//     PlcTask Inputs/GVL_iXlinker.EtherCAT_Master_EJxxxx.Beckhoff_EJ9xxx.A_0003_EJ9576_0000_0018.WcState.WcState <-> WcState/WcState
//     PlcTask Inputs/GVL_iXlinker.EtherCAT_Master_EJxxxx.Beckhoff_EJ9xxx.A_0003_EJ9576_0000_0018.WcState.InputToggle <-> WcState/InputToggle
//     PlcTask Inputs/GVL_iXlinker.EtherCAT_Master_EJxxxx.Beckhoff_EJ9xxx.A_0003_EJ9576_0000_0018.InfoData.AdsAddr <-> InfoData/AdsAddr
//     PlcTask Inputs/GVL_iXlinker.EtherCAT_Master_EJxxxx.Beckhoff_EJ9xxx.A_0003_EJ9576_0000_0018.InfoData.State <-> InfoData/State
//   PLC/PLC Instance <-> EtherCAT Master EJxxxx/Beckhoff EJ9xxx/A_0004(EJ9576-0000-0019)
//     PlcTask Inputs/GVL_iXlinker.EtherCAT_Master_EJxxxx.Beckhoff_EJ9xxx.A_0004_EJ9576_0000_0019.BCT_Inputs.Terminal_Overtemperature <-> BCT Inputs/Terminal Overtemperature
//     PlcTask Inputs/GVL_iXlinker.EtherCAT_Master_EJxxxx.Beckhoff_EJ9xxx.A_0004_EJ9576_0000_0019.BCT_Inputs.I2T_error <-> BCT Inputs/I2T error
//     PlcTask Inputs/GVL_iXlinker.EtherCAT_Master_EJxxxx.Beckhoff_EJ9xxx.A_0004_EJ9576_0000_0019.BCT_Inputs.I2T_warning <-> BCT Inputs/I2T warning
//     PlcTask Inputs/GVL_iXlinker.EtherCAT_Master_EJxxxx.Beckhoff_EJ9xxx.A_0004_EJ9576_0000_0019.BCT_Inputs.Overvoltage <-> BCT Inputs/Overvoltage
//     PlcTask Inputs/GVL_iXlinker.EtherCAT_Master_EJxxxx.Beckhoff_EJ9xxx.A_0004_EJ9576_0000_0019.BCT_Inputs.Undervoltage <-> BCT Inputs/Undervoltage
//     PlcTask Inputs/GVL_iXlinker.EtherCAT_Master_EJxxxx.Beckhoff_EJ9xxx.A_0004_EJ9576_0000_0019.BCT_Inputs.Chopper_on <-> BCT Inputs/Chopper on
//     PlcTask Inputs/GVL_iXlinker.EtherCAT_Master_EJxxxx.Beckhoff_EJ9xxx.A_0004_EJ9576_0000_0019.BCT_Inputs.Input_cycle_counter <-> BCT Inputs/Input cycle counter
//     PlcTask Inputs/GVL_iXlinker.EtherCAT_Master_EJxxxx.Beckhoff_EJ9xxx.A_0004_EJ9576_0000_0019.BCT_Inputs.DC_link_voltage <-> BCT Inputs/DC link voltage
//     PlcTask Inputs/GVL_iXlinker.EtherCAT_Master_EJxxxx.Beckhoff_EJ9xxx.A_0004_EJ9576_0000_0019.BCT_Inputs.Resistor_current <-> BCT Inputs/Resistor current
//     PlcTask Inputs/GVL_iXlinker.EtherCAT_Master_EJxxxx.Beckhoff_EJ9xxx.A_0004_EJ9576_0000_0019.BCT_Inputs.Duty_cylce <-> BCT Inputs/Duty cylce
//     PlcTask Inputs/GVL_iXlinker.EtherCAT_Master_EJxxxx.Beckhoff_EJ9xxx.A_0004_EJ9576_0000_0019.BCT_Inputs.I2T_load_factor <-> BCT Inputs/I2T load factor
//     PlcTask Inputs/GVL_iXlinker.EtherCAT_Master_EJxxxx.Beckhoff_EJ9xxx.A_0004_EJ9576_0000_0019.WcState.WcState <-> WcState/WcState
//     PlcTask Inputs/GVL_iXlinker.EtherCAT_Master_EJxxxx.Beckhoff_EJ9xxx.A_0004_EJ9576_0000_0019.WcState.InputToggle <-> WcState/InputToggle
//     PlcTask Inputs/GVL_iXlinker.EtherCAT_Master_EJxxxx.Beckhoff_EJ9xxx.A_0004_EJ9576_0000_0019.InfoData.AdsAddr <-> InfoData/AdsAddr
//     PlcTask Inputs/GVL_iXlinker.EtherCAT_Master_EJxxxx.Beckhoff_EJ9xxx.A_0004_EJ9576_0000_0019.InfoData.State <-> InfoData/State
//   PLC/PLC Instance <-> EtherCAT Master EJxxxx/Beckhoff EJ9xxx/A_0005(EJ9576-0000-0020)
//     PlcTask Inputs/GVL_iXlinker.EtherCAT_Master_EJxxxx.Beckhoff_EJ9xxx.A_0005_EJ9576_0000_0020.BCT_Inputs.Terminal_Overtemperature <-> BCT Inputs/Terminal Overtemperature
//     PlcTask Inputs/GVL_iXlinker.EtherCAT_Master_EJxxxx.Beckhoff_EJ9xxx.A_0005_EJ9576_0000_0020.BCT_Inputs.I2T_error <-> BCT Inputs/I2T error
//     PlcTask Inputs/GVL_iXlinker.EtherCAT_Master_EJxxxx.Beckhoff_EJ9xxx.A_0005_EJ9576_0000_0020.BCT_Inputs.I2T_warning <-> BCT Inputs/I2T warning
//     PlcTask Inputs/GVL_iXlinker.EtherCAT_Master_EJxxxx.Beckhoff_EJ9xxx.A_0005_EJ9576_0000_0020.BCT_Inputs.Overvoltage <-> BCT Inputs/Overvoltage
//     PlcTask Inputs/GVL_iXlinker.EtherCAT_Master_EJxxxx.Beckhoff_EJ9xxx.A_0005_EJ9576_0000_0020.BCT_Inputs.Undervoltage <-> BCT Inputs/Undervoltage
//     PlcTask Inputs/GVL_iXlinker.EtherCAT_Master_EJxxxx.Beckhoff_EJ9xxx.A_0005_EJ9576_0000_0020.BCT_Inputs.Chopper_on <-> BCT Inputs/Chopper on
//     PlcTask Inputs/GVL_iXlinker.EtherCAT_Master_EJxxxx.Beckhoff_EJ9xxx.A_0005_EJ9576_0000_0020.BCT_Inputs.Input_cycle_counter <-> BCT Inputs/Input cycle counter
//     PlcTask Inputs/GVL_iXlinker.EtherCAT_Master_EJxxxx.Beckhoff_EJ9xxx.A_0005_EJ9576_0000_0020.BCT_Inputs.DC_link_voltage <-> BCT Inputs/DC link voltage
//     PlcTask Inputs/GVL_iXlinker.EtherCAT_Master_EJxxxx.Beckhoff_EJ9xxx.A_0005_EJ9576_0000_0020.BCT_Inputs.Resistor_Current <-> BCT Inputs/Resistor Current
//     PlcTask Inputs/GVL_iXlinker.EtherCAT_Master_EJxxxx.Beckhoff_EJ9xxx.A_0005_EJ9576_0000_0020.BCT_Inputs.Duty_Cycle <-> BCT Inputs/Duty Cycle
//     PlcTask Inputs/GVL_iXlinker.EtherCAT_Master_EJxxxx.Beckhoff_EJ9xxx.A_0005_EJ9576_0000_0020.WcState.WcState <-> WcState/WcState
//     PlcTask Inputs/GVL_iXlinker.EtherCAT_Master_EJxxxx.Beckhoff_EJ9xxx.A_0005_EJ9576_0000_0020.WcState.InputToggle <-> WcState/InputToggle
//     PlcTask Inputs/GVL_iXlinker.EtherCAT_Master_EJxxxx.Beckhoff_EJ9xxx.A_0005_EJ9576_0000_0020.InfoData.AdsAddr <-> InfoData/AdsAddr
//     PlcTask Inputs/GVL_iXlinker.EtherCAT_Master_EJxxxx.Beckhoff_EJ9xxx.A_0005_EJ9576_0000_0020.InfoData.State <-> InfoData/State
//   PLC/PLC Instance <-> EtherCAT Master EJxxxx/Beckhoff EJ9xxx/A_0006(EJ9576-0000-0022)
//     PlcTask Inputs/GVL_iXlinker.EtherCAT_Master_EJxxxx.Beckhoff_EJ9xxx.A_0006_EJ9576_0000_0022.BCT_Inputs.Terminal_Overtemperature <-> BCT Inputs/Terminal Overtemperature
//     PlcTask Inputs/GVL_iXlinker.EtherCAT_Master_EJxxxx.Beckhoff_EJ9xxx.A_0006_EJ9576_0000_0022.BCT_Inputs.I2T_error <-> BCT Inputs/I2T error
//     PlcTask Inputs/GVL_iXlinker.EtherCAT_Master_EJxxxx.Beckhoff_EJ9xxx.A_0006_EJ9576_0000_0022.BCT_Inputs.I2T_warning <-> BCT Inputs/I2T warning
//     PlcTask Inputs/GVL_iXlinker.EtherCAT_Master_EJxxxx.Beckhoff_EJ9xxx.A_0006_EJ9576_0000_0022.BCT_Inputs.Overvoltage <-> BCT Inputs/Overvoltage
//     PlcTask Inputs/GVL_iXlinker.EtherCAT_Master_EJxxxx.Beckhoff_EJ9xxx.A_0006_EJ9576_0000_0022.BCT_Inputs.Undervoltage <-> BCT Inputs/Undervoltage
//     PlcTask Inputs/GVL_iXlinker.EtherCAT_Master_EJxxxx.Beckhoff_EJ9xxx.A_0006_EJ9576_0000_0022.BCT_Inputs.Chopper_on <-> BCT Inputs/Chopper on
//     PlcTask Inputs/GVL_iXlinker.EtherCAT_Master_EJxxxx.Beckhoff_EJ9xxx.A_0006_EJ9576_0000_0022.BCT_Inputs.Overcurrent_Protection <-> BCT Inputs/Overcurrent Protection
//     PlcTask Inputs/GVL_iXlinker.EtherCAT_Master_EJxxxx.Beckhoff_EJ9xxx.A_0006_EJ9576_0000_0022.BCT_Inputs.Input_cycle_counter <-> BCT Inputs/Input cycle counter
//     PlcTask Inputs/GVL_iXlinker.EtherCAT_Master_EJxxxx.Beckhoff_EJ9xxx.A_0006_EJ9576_0000_0022.BCT_Inputs.DC_link_voltage <-> BCT Inputs/DC link voltage
//     PlcTask Inputs/GVL_iXlinker.EtherCAT_Master_EJxxxx.Beckhoff_EJ9xxx.A_0006_EJ9576_0000_0022.BCT_Inputs.Resistor_Current <-> BCT Inputs/Resistor Current
//     PlcTask Inputs/GVL_iXlinker.EtherCAT_Master_EJxxxx.Beckhoff_EJ9xxx.A_0006_EJ9576_0000_0022.BCT_Inputs.Duty_Cycle <-> BCT Inputs/Duty Cycle
//     PlcTask Inputs/GVL_iXlinker.EtherCAT_Master_EJxxxx.Beckhoff_EJ9xxx.A_0006_EJ9576_0000_0022.WcState.WcState <-> WcState/WcState
//     PlcTask Inputs/GVL_iXlinker.EtherCAT_Master_EJxxxx.Beckhoff_EJ9xxx.A_0006_EJ9576_0000_0022.WcState.InputToggle <-> WcState/InputToggle
//     PlcTask Inputs/GVL_iXlinker.EtherCAT_Master_EJxxxx.Beckhoff_EJ9xxx.A_0006_EJ9576_0000_0022.InfoData.AdsAddr <-> InfoData/AdsAddr
//     PlcTask Inputs/GVL_iXlinker.EtherCAT_Master_EJxxxx.Beckhoff_EJ9xxx.A_0006_EJ9576_0000_0022.InfoData.State <-> InfoData/State
//   PLC/PLC Instance <-> EtherCAT Master EJxxxx/Beckhoff EJx9xx
//     PlcTask Inputs/GVL_iXlinker.EtherCAT_Master_EJxxxx.Beckhoff_EJx9xx.InfoData.State <-> InfoData/State
//   PLC/PLC Instance <-> EtherCAT Master EJxxxx/Beckhoff EJx9xx/Beckhoff EJx9xxEK1122
//     PlcTask Inputs/GVL_iXlinker.EtherCAT_Master_EJxxxx.Beckhoff_EJx9xx.Beckhoff_EJx9xxEK1122.InfoData.State <-> InfoData/State
//   PLC/PLC Instance <-> EtherCAT Master EJxxxx/Beckhoff EJx9xx/Beckhoff EJx9xxEK1122/Beckhoff EJx9xxsub EK1100
//     PlcTask Inputs/GVL_iXlinker.EtherCAT_Master_EJxxxx.Beckhoff_EJx9xx.Beckhoff_EJx9xxEK1122.Beckhoff_EJx9xxsub_EK1100.InfoData.State <-> InfoData/State
//   PLC/PLC Instance <-> EtherCAT Master EJxxxx/Beckhoff EJx9xx/A_0001(EJ1914-0000-0017)
//     PlcTask Inputs/GVL_iXlinker.EtherCAT_Master_EJxxxx.Beckhoff_EJx9xx.A_0001_EJ1914_0000_0017.Module_1_FSOE.FSoE_Inputs.FSOE/FSoE_Command <-> Module 1 (FSOE)/FSoE Inputs/FSOE/FSoE Command
//     PlcTask Inputs/GVL_iXlinker.EtherCAT_Master_EJxxxx.Beckhoff_EJx9xx.A_0001_EJ1914_0000_0017.Module_1_FSOE.FSoE_Inputs.FSOE/FSIN_Module_1_Channel_1_Input <-> Module 1 (FSOE)/FSoE Inputs/FSOE/FSIN Module 1.Channel 1.Input
//     PlcTask Inputs/GVL_iXlinker.EtherCAT_Master_EJxxxx.Beckhoff_EJx9xx.A_0001_EJ1914_0000_0017.Module_1_FSOE.FSoE_Inputs.FSOE/FSIN_Module_1_Channel_2_Input <-> Module 1 (FSOE)/FSoE Inputs/FSOE/FSIN Module 1.Channel 2.Input
//     PlcTask Inputs/GVL_iXlinker.EtherCAT_Master_EJxxxx.Beckhoff_EJx9xx.A_0001_EJ1914_0000_0017.Module_1_FSOE.FSoE_Inputs.FSOE/FSIN_Module_2_Channel_1_Input <-> Module 1 (FSOE)/FSoE Inputs/FSOE/FSIN Module 2.Channel 1.Input
//     PlcTask Inputs/GVL_iXlinker.EtherCAT_Master_EJxxxx.Beckhoff_EJx9xx.A_0001_EJ1914_0000_0017.Module_1_FSOE.FSoE_Inputs.FSOE/FSIN_Module_2_Channel_2_Input <-> Module 1 (FSOE)/FSoE Inputs/FSOE/FSIN Module 2.Channel 2.Input
//     PlcTask Inputs/GVL_iXlinker.EtherCAT_Master_EJxxxx.Beckhoff_EJx9xx.A_0001_EJ1914_0000_0017.Module_1_FSOE.FSoE_Inputs.FSOE/FSIN_Module_1_Module_Fault <-> Module 1 (FSOE)/FSoE Inputs/FSOE/FSIN Module 1.Module Fault
//     PlcTask Inputs/GVL_iXlinker.EtherCAT_Master_EJxxxx.Beckhoff_EJx9xx.A_0001_EJ1914_0000_0017.Module_1_FSOE.FSoE_Inputs.FSOE/FSIN_Module_2_Module_Fault <-> Module 1 (FSOE)/FSoE Inputs/FSOE/FSIN Module 2.Module Fault
//     PlcTask Inputs/GVL_iXlinker.EtherCAT_Master_EJxxxx.Beckhoff_EJx9xx.A_0001_EJ1914_0000_0017.Module_1_FSOE.FSoE_Inputs.FSOE/FSoE_CRC_000 <-> Module 1 (FSOE)/FSoE Inputs/FSOE/FSoE CRC 000
//     PlcTask Inputs/GVL_iXlinker.EtherCAT_Master_EJxxxx.Beckhoff_EJx9xx.A_0001_EJ1914_0000_0017.Module_1_FSOE.FSoE_Inputs.FSOE/FSoE_Connection_ID <-> Module 1 (FSOE)/FSoE Inputs/FSOE/FSoE Connection ID
//     PlcTask Outputs/GVL_iXlinker.EtherCAT_Master_EJxxxx.Beckhoff_EJx9xx.A_0001_EJ1914_0000_0017.Module_1_FSOE.FSoE_Outputs.FSOE/FSoE_Command <-> Module 1 (FSOE)/FSoE Outputs/FSOE/FSoE Command
//     PlcTask Outputs/GVL_iXlinker.EtherCAT_Master_EJxxxx.Beckhoff_EJx9xx.A_0001_EJ1914_0000_0017.Module_1_FSOE.FSoE_Outputs.FSOE/FSIN_Module_1_ErrAck <-> Module 1 (FSOE)/FSoE Outputs/FSOE/FSIN Module 1.ErrAck
//     PlcTask Outputs/GVL_iXlinker.EtherCAT_Master_EJxxxx.Beckhoff_EJx9xx.A_0001_EJ1914_0000_0017.Module_1_FSOE.FSoE_Outputs.FSOE/FSIN_Module_2_ErrAck <-> Module 1 (FSOE)/FSoE Outputs/FSOE/FSIN Module 2.ErrAck
//     PlcTask Outputs/GVL_iXlinker.EtherCAT_Master_EJxxxx.Beckhoff_EJx9xx.A_0001_EJ1914_0000_0017.Module_1_FSOE.FSoE_Outputs.FSOE/FSoE_CRC_000 <-> Module 1 (FSOE)/FSoE Outputs/FSOE/FSoE CRC 000
//     PlcTask Outputs/GVL_iXlinker.EtherCAT_Master_EJxxxx.Beckhoff_EJx9xx.A_0001_EJ1914_0000_0017.Module_1_FSOE.FSoE_Outputs.FSOE/FSoE_Connection_ID <-> Module 1 (FSOE)/FSoE Outputs/FSOE/FSoE Connection ID
//     PlcTask Inputs/GVL_iXlinker.EtherCAT_Master_EJxxxx.Beckhoff_EJx9xx.A_0001_EJ1914_0000_0017.Module_2_DEVICEIO.FIELDVOLTAGE_Field_Voltage_Status.Fieldvoltage_Underrange <-> Module 2 (DEVICEIO)/FIELDVOLTAGE Field Voltage Status/Fieldvoltage Underrange
//     PlcTask Inputs/GVL_iXlinker.EtherCAT_Master_EJxxxx.Beckhoff_EJx9xx.A_0001_EJ1914_0000_0017.Module_2_DEVICEIO.FIELDVOLTAGE_Field_Voltage_Status.Fieldvoltage_Overrange <-> Module 2 (DEVICEIO)/FIELDVOLTAGE Field Voltage Status/Fieldvoltage Overrange
//     PlcTask Inputs/GVL_iXlinker.EtherCAT_Master_EJxxxx.Beckhoff_EJx9xx.A_0001_EJ1914_0000_0017.Module_3_FSLOGIC.FSLOGIC_Inputs.Safe_Logic_State <-> Module 3 (FSLOGIC)/FSLOGIC Inputs/Safe Logic State
//     PlcTask Inputs/GVL_iXlinker.EtherCAT_Master_EJxxxx.Beckhoff_EJx9xx.A_0001_EJ1914_0000_0017.Module_3_FSLOGIC.FSLOGIC_Inputs.Cycle_Counter <-> Module 3 (FSLOGIC)/FSLOGIC Inputs/Cycle Counter
//     PlcTask Inputs/GVL_iXlinker.EtherCAT_Master_EJxxxx.Beckhoff_EJx9xx.A_0001_EJ1914_0000_0017.WcState.WcState <-> WcState/WcState
//     PlcTask Inputs/GVL_iXlinker.EtherCAT_Master_EJxxxx.Beckhoff_EJx9xx.A_0001_EJ1914_0000_0017.WcState.InputToggle <-> WcState/InputToggle
//     PlcTask Inputs/GVL_iXlinker.EtherCAT_Master_EJxxxx.Beckhoff_EJx9xx.A_0001_EJ1914_0000_0017.InfoData.AdsAddr <-> InfoData/AdsAddr
//     PlcTask Inputs/GVL_iXlinker.EtherCAT_Master_EJxxxx.Beckhoff_EJx9xx.A_0001_EJ1914_0000_0017.InfoData.State <-> InfoData/State
//   PLC/PLC Instance <-> EtherCAT Master EJxxxx/Beckhoff EJx9xx/A_0002(EJ1914-0000-0018)
//     PlcTask Inputs/GVL_iXlinker.EtherCAT_Master_EJxxxx.Beckhoff_EJx9xx.A_0002_EJ1914_0000_0018.Module_1_FSOE.FSoE_Inputs.FSOE/FSoE_Command <-> Module 1 (FSOE)/FSoE Inputs/FSOE/FSoE Command
//     PlcTask Inputs/GVL_iXlinker.EtherCAT_Master_EJxxxx.Beckhoff_EJx9xx.A_0002_EJ1914_0000_0018.Module_1_FSOE.FSoE_Inputs.FSOE/FSIN_Module_1_Channel_1_Input <-> Module 1 (FSOE)/FSoE Inputs/FSOE/FSIN Module 1.Channel 1.Input
//     PlcTask Inputs/GVL_iXlinker.EtherCAT_Master_EJxxxx.Beckhoff_EJx9xx.A_0002_EJ1914_0000_0018.Module_1_FSOE.FSoE_Inputs.FSOE/FSIN_Module_1_Channel_2_Input <-> Module 1 (FSOE)/FSoE Inputs/FSOE/FSIN Module 1.Channel 2.Input
//     PlcTask Inputs/GVL_iXlinker.EtherCAT_Master_EJxxxx.Beckhoff_EJx9xx.A_0002_EJ1914_0000_0018.Module_1_FSOE.FSoE_Inputs.FSOE/FSIN_Module_2_Channel_1_Input <-> Module 1 (FSOE)/FSoE Inputs/FSOE/FSIN Module 2.Channel 1.Input
//     PlcTask Inputs/GVL_iXlinker.EtherCAT_Master_EJxxxx.Beckhoff_EJx9xx.A_0002_EJ1914_0000_0018.Module_1_FSOE.FSoE_Inputs.FSOE/FSIN_Module_2_Channel_2_Input <-> Module 1 (FSOE)/FSoE Inputs/FSOE/FSIN Module 2.Channel 2.Input
//     PlcTask Inputs/GVL_iXlinker.EtherCAT_Master_EJxxxx.Beckhoff_EJx9xx.A_0002_EJ1914_0000_0018.Module_1_FSOE.FSoE_Inputs.FSOE/FSIN_Module_1_Module_Fault <-> Module 1 (FSOE)/FSoE Inputs/FSOE/FSIN Module 1.Module Fault
//     PlcTask Inputs/GVL_iXlinker.EtherCAT_Master_EJxxxx.Beckhoff_EJx9xx.A_0002_EJ1914_0000_0018.Module_1_FSOE.FSoE_Inputs.FSOE/FSIN_Module_2_Module_Fault <-> Module 1 (FSOE)/FSoE Inputs/FSOE/FSIN Module 2.Module Fault
//     PlcTask Inputs/GVL_iXlinker.EtherCAT_Master_EJxxxx.Beckhoff_EJx9xx.A_0002_EJ1914_0000_0018.Module_1_FSOE.FSoE_Inputs.FSOE/FSoE_CRC_000 <-> Module 1 (FSOE)/FSoE Inputs/FSOE/FSoE CRC 000
//     PlcTask Inputs/GVL_iXlinker.EtherCAT_Master_EJxxxx.Beckhoff_EJx9xx.A_0002_EJ1914_0000_0018.Module_1_FSOE.FSoE_Inputs.FSOE/FSoE_Connection_ID <-> Module 1 (FSOE)/FSoE Inputs/FSOE/FSoE Connection ID
//     PlcTask Outputs/GVL_iXlinker.EtherCAT_Master_EJxxxx.Beckhoff_EJx9xx.A_0002_EJ1914_0000_0018.Module_1_FSOE.FSoE_Outputs.FSOE/FSoE_Command <-> Module 1 (FSOE)/FSoE Outputs/FSOE/FSoE Command
//     PlcTask Outputs/GVL_iXlinker.EtherCAT_Master_EJxxxx.Beckhoff_EJx9xx.A_0002_EJ1914_0000_0018.Module_1_FSOE.FSoE_Outputs.FSOE/FSIN_Module_1_ErrAck <-> Module 1 (FSOE)/FSoE Outputs/FSOE/FSIN Module 1.ErrAck
//     PlcTask Outputs/GVL_iXlinker.EtherCAT_Master_EJxxxx.Beckhoff_EJx9xx.A_0002_EJ1914_0000_0018.Module_1_FSOE.FSoE_Outputs.FSOE/FSIN_Module_2_ErrAck <-> Module 1 (FSOE)/FSoE Outputs/FSOE/FSIN Module 2.ErrAck
//     PlcTask Outputs/GVL_iXlinker.EtherCAT_Master_EJxxxx.Beckhoff_EJx9xx.A_0002_EJ1914_0000_0018.Module_1_FSOE.FSoE_Outputs.FSOE/FSoE_CRC_000 <-> Module 1 (FSOE)/FSoE Outputs/FSOE/FSoE CRC 000
//     PlcTask Outputs/GVL_iXlinker.EtherCAT_Master_EJxxxx.Beckhoff_EJx9xx.A_0002_EJ1914_0000_0018.Module_1_FSOE.FSoE_Outputs.FSOE/FSoE_Connection_ID <-> Module 1 (FSOE)/FSoE Outputs/FSOE/FSoE Connection ID
//     PlcTask Inputs/GVL_iXlinker.EtherCAT_Master_EJxxxx.Beckhoff_EJx9xx.A_0002_EJ1914_0000_0018.Module_2_DEVICEIO.FIELDVOLTAGE_Field_Voltage_Status.Fieldvoltage_Underrange <-> Module 2 (DEVICEIO)/FIELDVOLTAGE Field Voltage Status/Fieldvoltage Underrange
//     PlcTask Inputs/GVL_iXlinker.EtherCAT_Master_EJxxxx.Beckhoff_EJx9xx.A_0002_EJ1914_0000_0018.Module_2_DEVICEIO.FIELDVOLTAGE_Field_Voltage_Status.Fieldvoltage_Overrange <-> Module 2 (DEVICEIO)/FIELDVOLTAGE Field Voltage Status/Fieldvoltage Overrange
//     PlcTask Inputs/GVL_iXlinker.EtherCAT_Master_EJxxxx.Beckhoff_EJx9xx.A_0002_EJ1914_0000_0018.Module_3_FSLOGIC.FSLOGIC_Inputs.Safe_Logic_State <-> Module 3 (FSLOGIC)/FSLOGIC Inputs/Safe Logic State
//     PlcTask Inputs/GVL_iXlinker.EtherCAT_Master_EJxxxx.Beckhoff_EJx9xx.A_0002_EJ1914_0000_0018.Module_3_FSLOGIC.FSLOGIC_Inputs.Cycle_Counter <-> Module 3 (FSLOGIC)/FSLOGIC Inputs/Cycle Counter
//     PlcTask Inputs/GVL_iXlinker.EtherCAT_Master_EJxxxx.Beckhoff_EJx9xx.A_0002_EJ1914_0000_0018.WcState.WcState <-> WcState/WcState
//     PlcTask Inputs/GVL_iXlinker.EtherCAT_Master_EJxxxx.Beckhoff_EJx9xx.A_0002_EJ1914_0000_0018.WcState.InputToggle <-> WcState/InputToggle
//     PlcTask Inputs/GVL_iXlinker.EtherCAT_Master_EJxxxx.Beckhoff_EJx9xx.A_0002_EJ1914_0000_0018.InfoData.AdsAddr <-> InfoData/AdsAddr
//     PlcTask Inputs/GVL_iXlinker.EtherCAT_Master_EJxxxx.Beckhoff_EJx9xx.A_0002_EJ1914_0000_0018.InfoData.State <-> InfoData/State
//   PLC/PLC Instance <-> EtherCAT Master EJxxxx/Beckhoff EJx9xx/A_0003(EJ1918-0000-0017)
//     PlcTask Inputs/GVL_iXlinker.EtherCAT_Master_EJxxxx.Beckhoff_EJx9xx.A_0003_EJ1918_0000_0017.Module_1_FSOE.FSoE_Inputs.FSOE/FSoE_Command <-> Module 1 (FSOE)/FSoE Inputs/FSOE/FSoE Command
//     PlcTask Inputs/GVL_iXlinker.EtherCAT_Master_EJxxxx.Beckhoff_EJx9xx.A_0003_EJ1918_0000_0017.Module_1_FSOE.FSoE_Inputs.FSOE/FSIN_Module_1_Channel_1_Input <-> Module 1 (FSOE)/FSoE Inputs/FSOE/FSIN Module 1.Channel 1.Input
//     PlcTask Inputs/GVL_iXlinker.EtherCAT_Master_EJxxxx.Beckhoff_EJx9xx.A_0003_EJ1918_0000_0017.Module_1_FSOE.FSoE_Inputs.FSOE/FSIN_Module_1_Channel_2_Input <-> Module 1 (FSOE)/FSoE Inputs/FSOE/FSIN Module 1.Channel 2.Input
//     PlcTask Inputs/GVL_iXlinker.EtherCAT_Master_EJxxxx.Beckhoff_EJx9xx.A_0003_EJ1918_0000_0017.Module_1_FSOE.FSoE_Inputs.FSOE/FSIN_Module_2_Channel_1_Input <-> Module 1 (FSOE)/FSoE Inputs/FSOE/FSIN Module 2.Channel 1.Input
//     PlcTask Inputs/GVL_iXlinker.EtherCAT_Master_EJxxxx.Beckhoff_EJx9xx.A_0003_EJ1918_0000_0017.Module_1_FSOE.FSoE_Inputs.FSOE/FSIN_Module_2_Channel_2_Input <-> Module 1 (FSOE)/FSoE Inputs/FSOE/FSIN Module 2.Channel 2.Input
//     PlcTask Inputs/GVL_iXlinker.EtherCAT_Master_EJxxxx.Beckhoff_EJx9xx.A_0003_EJ1918_0000_0017.Module_1_FSOE.FSoE_Inputs.FSOE/FSIN_Module_3_Channel_1_Input <-> Module 1 (FSOE)/FSoE Inputs/FSOE/FSIN Module 3.Channel 1.Input
//     PlcTask Inputs/GVL_iXlinker.EtherCAT_Master_EJxxxx.Beckhoff_EJx9xx.A_0003_EJ1918_0000_0017.Module_1_FSOE.FSoE_Inputs.FSOE/FSIN_Module_3_Channel_2_Input <-> Module 1 (FSOE)/FSoE Inputs/FSOE/FSIN Module 3.Channel 2.Input
//     PlcTask Inputs/GVL_iXlinker.EtherCAT_Master_EJxxxx.Beckhoff_EJx9xx.A_0003_EJ1918_0000_0017.Module_1_FSOE.FSoE_Inputs.FSOE/FSIN_Module_4_Channel_1_Input <-> Module 1 (FSOE)/FSoE Inputs/FSOE/FSIN Module 4.Channel 1.Input
//     PlcTask Inputs/GVL_iXlinker.EtherCAT_Master_EJxxxx.Beckhoff_EJx9xx.A_0003_EJ1918_0000_0017.Module_1_FSOE.FSoE_Inputs.FSOE/FSIN_Module_4_Channel_2_Input <-> Module 1 (FSOE)/FSoE Inputs/FSOE/FSIN Module 4.Channel 2.Input
//     PlcTask Inputs/GVL_iXlinker.EtherCAT_Master_EJxxxx.Beckhoff_EJx9xx.A_0003_EJ1918_0000_0017.Module_1_FSOE.FSoE_Inputs.FSOE/FSIN_Module_1_Module_Fault <-> Module 1 (FSOE)/FSoE Inputs/FSOE/FSIN Module 1.Module Fault
//     PlcTask Inputs/GVL_iXlinker.EtherCAT_Master_EJxxxx.Beckhoff_EJx9xx.A_0003_EJ1918_0000_0017.Module_1_FSOE.FSoE_Inputs.FSOE/FSIN_Module_2_Module_Fault <-> Module 1 (FSOE)/FSoE Inputs/FSOE/FSIN Module 2.Module Fault
//     PlcTask Inputs/GVL_iXlinker.EtherCAT_Master_EJxxxx.Beckhoff_EJx9xx.A_0003_EJ1918_0000_0017.Module_1_FSOE.FSoE_Inputs.FSOE/FSIN_Module_3_Module_Fault <-> Module 1 (FSOE)/FSoE Inputs/FSOE/FSIN Module 3.Module Fault
//     PlcTask Inputs/GVL_iXlinker.EtherCAT_Master_EJxxxx.Beckhoff_EJx9xx.A_0003_EJ1918_0000_0017.Module_1_FSOE.FSoE_Inputs.FSOE/FSIN_Module_4_Module_Fault <-> Module 1 (FSOE)/FSoE Inputs/FSOE/FSIN Module 4.Module Fault
//     PlcTask Inputs/GVL_iXlinker.EtherCAT_Master_EJxxxx.Beckhoff_EJx9xx.A_0003_EJ1918_0000_0017.Module_1_FSOE.FSoE_Inputs.FSOE/FSoE_CRC_000 <-> Module 1 (FSOE)/FSoE Inputs/FSOE/FSoE CRC 000
//     PlcTask Inputs/GVL_iXlinker.EtherCAT_Master_EJxxxx.Beckhoff_EJx9xx.A_0003_EJ1918_0000_0017.Module_1_FSOE.FSoE_Inputs.FSOE/FSoE_Connection_ID <-> Module 1 (FSOE)/FSoE Inputs/FSOE/FSoE Connection ID
//     PlcTask Outputs/GVL_iXlinker.EtherCAT_Master_EJxxxx.Beckhoff_EJx9xx.A_0003_EJ1918_0000_0017.Module_1_FSOE.FSoE_Outputs.FSOE/FSoE_Command <-> Module 1 (FSOE)/FSoE Outputs/FSOE/FSoE Command
//     PlcTask Outputs/GVL_iXlinker.EtherCAT_Master_EJxxxx.Beckhoff_EJx9xx.A_0003_EJ1918_0000_0017.Module_1_FSOE.FSoE_Outputs.FSOE/FSIN_Module_1_ErrAck <-> Module 1 (FSOE)/FSoE Outputs/FSOE/FSIN Module 1.ErrAck
//     PlcTask Outputs/GVL_iXlinker.EtherCAT_Master_EJxxxx.Beckhoff_EJx9xx.A_0003_EJ1918_0000_0017.Module_1_FSOE.FSoE_Outputs.FSOE/FSIN_Module_2_ErrAck <-> Module 1 (FSOE)/FSoE Outputs/FSOE/FSIN Module 2.ErrAck
//     PlcTask Outputs/GVL_iXlinker.EtherCAT_Master_EJxxxx.Beckhoff_EJx9xx.A_0003_EJ1918_0000_0017.Module_1_FSOE.FSoE_Outputs.FSOE/FSIN_Module_3_ErrAck <-> Module 1 (FSOE)/FSoE Outputs/FSOE/FSIN Module 3.ErrAck
//     PlcTask Outputs/GVL_iXlinker.EtherCAT_Master_EJxxxx.Beckhoff_EJx9xx.A_0003_EJ1918_0000_0017.Module_1_FSOE.FSoE_Outputs.FSOE/FSIN_Module_4_ErrAck <-> Module 1 (FSOE)/FSoE Outputs/FSOE/FSIN Module 4.ErrAck
//     PlcTask Outputs/GVL_iXlinker.EtherCAT_Master_EJxxxx.Beckhoff_EJx9xx.A_0003_EJ1918_0000_0017.Module_1_FSOE.FSoE_Outputs.FSOE/FSoE_CRC_000 <-> Module 1 (FSOE)/FSoE Outputs/FSOE/FSoE CRC 000
//     PlcTask Outputs/GVL_iXlinker.EtherCAT_Master_EJxxxx.Beckhoff_EJx9xx.A_0003_EJ1918_0000_0017.Module_1_FSOE.FSoE_Outputs.FSOE/FSoE_Connection_ID <-> Module 1 (FSOE)/FSoE Outputs/FSOE/FSoE Connection ID
//     PlcTask Inputs/GVL_iXlinker.EtherCAT_Master_EJxxxx.Beckhoff_EJx9xx.A_0003_EJ1918_0000_0017.Module_2_DEVICEIO.FIELDVOLTAGE_Field_Voltage_Status.Fieldvoltage_Underrange <-> Module 2 (DEVICEIO)/FIELDVOLTAGE Field Voltage Status/Fieldvoltage Underrange
//     PlcTask Inputs/GVL_iXlinker.EtherCAT_Master_EJxxxx.Beckhoff_EJx9xx.A_0003_EJ1918_0000_0017.Module_2_DEVICEIO.FIELDVOLTAGE_Field_Voltage_Status.Fieldvoltage_Overrange <-> Module 2 (DEVICEIO)/FIELDVOLTAGE Field Voltage Status/Fieldvoltage Overrange
//     PlcTask Inputs/GVL_iXlinker.EtherCAT_Master_EJxxxx.Beckhoff_EJx9xx.A_0003_EJ1918_0000_0017.Module_3_FSLOGIC.FSLOGIC_Inputs.Safe_Logic_State <-> Module 3 (FSLOGIC)/FSLOGIC Inputs/Safe Logic State
//     PlcTask Inputs/GVL_iXlinker.EtherCAT_Master_EJxxxx.Beckhoff_EJx9xx.A_0003_EJ1918_0000_0017.Module_3_FSLOGIC.FSLOGIC_Inputs.Cycle_Counter <-> Module 3 (FSLOGIC)/FSLOGIC Inputs/Cycle Counter
//     PlcTask Inputs/GVL_iXlinker.EtherCAT_Master_EJxxxx.Beckhoff_EJx9xx.A_0003_EJ1918_0000_0017.WcState.WcState <-> WcState/WcState
//     PlcTask Inputs/GVL_iXlinker.EtherCAT_Master_EJxxxx.Beckhoff_EJx9xx.A_0003_EJ1918_0000_0017.WcState.InputToggle <-> WcState/InputToggle
//     PlcTask Inputs/GVL_iXlinker.EtherCAT_Master_EJxxxx.Beckhoff_EJx9xx.A_0003_EJ1918_0000_0017.InfoData.AdsAddr <-> InfoData/AdsAddr
//     PlcTask Inputs/GVL_iXlinker.EtherCAT_Master_EJxxxx.Beckhoff_EJx9xx.A_0003_EJ1918_0000_0017.InfoData.State <-> InfoData/State
//   PLC/PLC Instance <-> EtherCAT Master EJxxxx/Beckhoff EJx9xx/A_0004(EJ1918-0000-0018)
//     PlcTask Inputs/GVL_iXlinker.EtherCAT_Master_EJxxxx.Beckhoff_EJx9xx.A_0004_EJ1918_0000_0018.Module_1_FSOE.FSoE_Inputs.FSOE/FSoE_Command <-> Module 1 (FSOE)/FSoE Inputs/FSOE/FSoE Command
//     PlcTask Inputs/GVL_iXlinker.EtherCAT_Master_EJxxxx.Beckhoff_EJx9xx.A_0004_EJ1918_0000_0018.Module_1_FSOE.FSoE_Inputs.FSOE/FSIN_Module_1_Channel_1_Input <-> Module 1 (FSOE)/FSoE Inputs/FSOE/FSIN Module 1.Channel 1.Input
//     PlcTask Inputs/GVL_iXlinker.EtherCAT_Master_EJxxxx.Beckhoff_EJx9xx.A_0004_EJ1918_0000_0018.Module_1_FSOE.FSoE_Inputs.FSOE/FSIN_Module_1_Channel_2_Input <-> Module 1 (FSOE)/FSoE Inputs/FSOE/FSIN Module 1.Channel 2.Input
//     PlcTask Inputs/GVL_iXlinker.EtherCAT_Master_EJxxxx.Beckhoff_EJx9xx.A_0004_EJ1918_0000_0018.Module_1_FSOE.FSoE_Inputs.FSOE/FSIN_Module_2_Channel_1_Input <-> Module 1 (FSOE)/FSoE Inputs/FSOE/FSIN Module 2.Channel 1.Input
//     PlcTask Inputs/GVL_iXlinker.EtherCAT_Master_EJxxxx.Beckhoff_EJx9xx.A_0004_EJ1918_0000_0018.Module_1_FSOE.FSoE_Inputs.FSOE/FSIN_Module_2_Channel_2_Input <-> Module 1 (FSOE)/FSoE Inputs/FSOE/FSIN Module 2.Channel 2.Input
//     PlcTask Inputs/GVL_iXlinker.EtherCAT_Master_EJxxxx.Beckhoff_EJx9xx.A_0004_EJ1918_0000_0018.Module_1_FSOE.FSoE_Inputs.FSOE/FSIN_Module_3_Channel_1_Input <-> Module 1 (FSOE)/FSoE Inputs/FSOE/FSIN Module 3.Channel 1.Input
//     PlcTask Inputs/GVL_iXlinker.EtherCAT_Master_EJxxxx.Beckhoff_EJx9xx.A_0004_EJ1918_0000_0018.Module_1_FSOE.FSoE_Inputs.FSOE/FSIN_Module_3_Channel_2_Input <-> Module 1 (FSOE)/FSoE Inputs/FSOE/FSIN Module 3.Channel 2.Input
//     PlcTask Inputs/GVL_iXlinker.EtherCAT_Master_EJxxxx.Beckhoff_EJx9xx.A_0004_EJ1918_0000_0018.Module_1_FSOE.FSoE_Inputs.FSOE/FSIN_Module_4_Channel_1_Input <-> Module 1 (FSOE)/FSoE Inputs/FSOE/FSIN Module 4.Channel 1.Input
//     PlcTask Inputs/GVL_iXlinker.EtherCAT_Master_EJxxxx.Beckhoff_EJx9xx.A_0004_EJ1918_0000_0018.Module_1_FSOE.FSoE_Inputs.FSOE/FSIN_Module_4_Channel_2_Input <-> Module 1 (FSOE)/FSoE Inputs/FSOE/FSIN Module 4.Channel 2.Input
//     PlcTask Inputs/GVL_iXlinker.EtherCAT_Master_EJxxxx.Beckhoff_EJx9xx.A_0004_EJ1918_0000_0018.Module_1_FSOE.FSoE_Inputs.FSOE/FSIN_Module_1_Module_Fault <-> Module 1 (FSOE)/FSoE Inputs/FSOE/FSIN Module 1.Module Fault
//     PlcTask Inputs/GVL_iXlinker.EtherCAT_Master_EJxxxx.Beckhoff_EJx9xx.A_0004_EJ1918_0000_0018.Module_1_FSOE.FSoE_Inputs.FSOE/FSIN_Module_2_Module_Fault <-> Module 1 (FSOE)/FSoE Inputs/FSOE/FSIN Module 2.Module Fault
//     PlcTask Inputs/GVL_iXlinker.EtherCAT_Master_EJxxxx.Beckhoff_EJx9xx.A_0004_EJ1918_0000_0018.Module_1_FSOE.FSoE_Inputs.FSOE/FSIN_Module_3_Module_Fault <-> Module 1 (FSOE)/FSoE Inputs/FSOE/FSIN Module 3.Module Fault
//     PlcTask Inputs/GVL_iXlinker.EtherCAT_Master_EJxxxx.Beckhoff_EJx9xx.A_0004_EJ1918_0000_0018.Module_1_FSOE.FSoE_Inputs.FSOE/FSIN_Module_4_Module_Fault <-> Module 1 (FSOE)/FSoE Inputs/FSOE/FSIN Module 4.Module Fault
//     PlcTask Inputs/GVL_iXlinker.EtherCAT_Master_EJxxxx.Beckhoff_EJx9xx.A_0004_EJ1918_0000_0018.Module_1_FSOE.FSoE_Inputs.FSOE/FSoE_CRC_000 <-> Module 1 (FSOE)/FSoE Inputs/FSOE/FSoE CRC 000
//     PlcTask Inputs/GVL_iXlinker.EtherCAT_Master_EJxxxx.Beckhoff_EJx9xx.A_0004_EJ1918_0000_0018.Module_1_FSOE.FSoE_Inputs.FSOE/FSoE_Connection_ID <-> Module 1 (FSOE)/FSoE Inputs/FSOE/FSoE Connection ID
//     PlcTask Outputs/GVL_iXlinker.EtherCAT_Master_EJxxxx.Beckhoff_EJx9xx.A_0004_EJ1918_0000_0018.Module_1_FSOE.FSoE_Outputs.FSOE/FSoE_Command <-> Module 1 (FSOE)/FSoE Outputs/FSOE/FSoE Command
//     PlcTask Outputs/GVL_iXlinker.EtherCAT_Master_EJxxxx.Beckhoff_EJx9xx.A_0004_EJ1918_0000_0018.Module_1_FSOE.FSoE_Outputs.FSOE/FSIN_Module_1_ErrAck <-> Module 1 (FSOE)/FSoE Outputs/FSOE/FSIN Module 1.ErrAck
//     PlcTask Outputs/GVL_iXlinker.EtherCAT_Master_EJxxxx.Beckhoff_EJx9xx.A_0004_EJ1918_0000_0018.Module_1_FSOE.FSoE_Outputs.FSOE/FSIN_Module_2_ErrAck <-> Module 1 (FSOE)/FSoE Outputs/FSOE/FSIN Module 2.ErrAck
//     PlcTask Outputs/GVL_iXlinker.EtherCAT_Master_EJxxxx.Beckhoff_EJx9xx.A_0004_EJ1918_0000_0018.Module_1_FSOE.FSoE_Outputs.FSOE/FSIN_Module_3_ErrAck <-> Module 1 (FSOE)/FSoE Outputs/FSOE/FSIN Module 3.ErrAck
//     PlcTask Outputs/GVL_iXlinker.EtherCAT_Master_EJxxxx.Beckhoff_EJx9xx.A_0004_EJ1918_0000_0018.Module_1_FSOE.FSoE_Outputs.FSOE/FSIN_Module_4_ErrAck <-> Module 1 (FSOE)/FSoE Outputs/FSOE/FSIN Module 4.ErrAck
//     PlcTask Outputs/GVL_iXlinker.EtherCAT_Master_EJxxxx.Beckhoff_EJx9xx.A_0004_EJ1918_0000_0018.Module_1_FSOE.FSoE_Outputs.FSOE/FSoE_CRC_000 <-> Module 1 (FSOE)/FSoE Outputs/FSOE/FSoE CRC 000
//     PlcTask Outputs/GVL_iXlinker.EtherCAT_Master_EJxxxx.Beckhoff_EJx9xx.A_0004_EJ1918_0000_0018.Module_1_FSOE.FSoE_Outputs.FSOE/FSoE_Connection_ID <-> Module 1 (FSOE)/FSoE Outputs/FSOE/FSoE Connection ID
//     PlcTask Inputs/GVL_iXlinker.EtherCAT_Master_EJxxxx.Beckhoff_EJx9xx.A_0004_EJ1918_0000_0018.Module_2_DEVICEIO.FIELDVOLTAGE_Field_Voltage_Status.Fieldvoltage_Underrange <-> Module 2 (DEVICEIO)/FIELDVOLTAGE Field Voltage Status/Fieldvoltage Underrange
//     PlcTask Inputs/GVL_iXlinker.EtherCAT_Master_EJxxxx.Beckhoff_EJx9xx.A_0004_EJ1918_0000_0018.Module_2_DEVICEIO.FIELDVOLTAGE_Field_Voltage_Status.Fieldvoltage_Overrange <-> Module 2 (DEVICEIO)/FIELDVOLTAGE Field Voltage Status/Fieldvoltage Overrange
//     PlcTask Inputs/GVL_iXlinker.EtherCAT_Master_EJxxxx.Beckhoff_EJx9xx.A_0004_EJ1918_0000_0018.Module_3_FSLOGIC.FSLOGIC_Inputs.Safe_Logic_State <-> Module 3 (FSLOGIC)/FSLOGIC Inputs/Safe Logic State
//     PlcTask Inputs/GVL_iXlinker.EtherCAT_Master_EJxxxx.Beckhoff_EJx9xx.A_0004_EJ1918_0000_0018.Module_3_FSLOGIC.FSLOGIC_Inputs.Cycle_Counter <-> Module 3 (FSLOGIC)/FSLOGIC Inputs/Cycle Counter
//     PlcTask Inputs/GVL_iXlinker.EtherCAT_Master_EJxxxx.Beckhoff_EJx9xx.A_0004_EJ1918_0000_0018.WcState.WcState <-> WcState/WcState
//     PlcTask Inputs/GVL_iXlinker.EtherCAT_Master_EJxxxx.Beckhoff_EJx9xx.A_0004_EJ1918_0000_0018.WcState.InputToggle <-> WcState/InputToggle
//     PlcTask Inputs/GVL_iXlinker.EtherCAT_Master_EJxxxx.Beckhoff_EJx9xx.A_0004_EJ1918_0000_0018.InfoData.AdsAddr <-> InfoData/AdsAddr
//     PlcTask Inputs/GVL_iXlinker.EtherCAT_Master_EJxxxx.Beckhoff_EJx9xx.A_0004_EJ1918_0000_0018.InfoData.State <-> InfoData/State
//   PLC/PLC Instance <-> EtherCAT Master EJxxxx/Beckhoff EJx9xx/A_0005(EJ1957-0000-0017)
//     PlcTask Inputs/GVL_iXlinker.EtherCAT_Master_EJxxxx.Beckhoff_EJx9xx.A_0005_EJ1957_0000_0017.Module_1_FSOE.FSoE_Inputs.FSOE/FSoE_Command <-> Module 1 (FSOE)/FSoE Inputs/FSOE/FSoE Command
//     PlcTask Inputs/GVL_iXlinker.EtherCAT_Master_EJxxxx.Beckhoff_EJx9xx.A_0005_EJ1957_0000_0017.Module_1_FSOE.FSoE_Inputs.FSOE/FSOUT_Module_Module_Fault <-> Module 1 (FSOE)/FSoE Inputs/FSOE/FSOUT Module.Module Fault
//     PlcTask Inputs/GVL_iXlinker.EtherCAT_Master_EJxxxx.Beckhoff_EJx9xx.A_0005_EJ1957_0000_0017.Module_1_FSOE.FSoE_Inputs.FSOE/FSIN_Module_1_Channel_1_Input <-> Module 1 (FSOE)/FSoE Inputs/FSOE/FSIN Module 1.Channel 1.Input
//     PlcTask Inputs/GVL_iXlinker.EtherCAT_Master_EJxxxx.Beckhoff_EJx9xx.A_0005_EJ1957_0000_0017.Module_1_FSOE.FSoE_Inputs.FSOE/FSIN_Module_1_Channel_2_Input <-> Module 1 (FSOE)/FSoE Inputs/FSOE/FSIN Module 1.Channel 2.Input
//     PlcTask Inputs/GVL_iXlinker.EtherCAT_Master_EJxxxx.Beckhoff_EJx9xx.A_0005_EJ1957_0000_0017.Module_1_FSOE.FSoE_Inputs.FSOE/FSIN_Module_2_Channel_1_Input <-> Module 1 (FSOE)/FSoE Inputs/FSOE/FSIN Module 2.Channel 1.Input
//     PlcTask Inputs/GVL_iXlinker.EtherCAT_Master_EJxxxx.Beckhoff_EJx9xx.A_0005_EJ1957_0000_0017.Module_1_FSOE.FSoE_Inputs.FSOE/FSIN_Module_2_Channel_2_Input <-> Module 1 (FSOE)/FSoE Inputs/FSOE/FSIN Module 2.Channel 2.Input
//     PlcTask Inputs/GVL_iXlinker.EtherCAT_Master_EJxxxx.Beckhoff_EJx9xx.A_0005_EJ1957_0000_0017.Module_1_FSOE.FSoE_Inputs.FSOE/FSIN_Module_3_Channel_1_Input <-> Module 1 (FSOE)/FSoE Inputs/FSOE/FSIN Module 3.Channel 1.Input
//     PlcTask Inputs/GVL_iXlinker.EtherCAT_Master_EJxxxx.Beckhoff_EJx9xx.A_0005_EJ1957_0000_0017.Module_1_FSOE.FSoE_Inputs.FSOE/FSIN_Module_3_Channel_2_Input <-> Module 1 (FSOE)/FSoE Inputs/FSOE/FSIN Module 3.Channel 2.Input
//     PlcTask Inputs/GVL_iXlinker.EtherCAT_Master_EJxxxx.Beckhoff_EJx9xx.A_0005_EJ1957_0000_0017.Module_1_FSOE.FSoE_Inputs.FSOE/FSIN_Module_4_Channel_1_Input <-> Module 1 (FSOE)/FSoE Inputs/FSOE/FSIN Module 4.Channel 1.Input
//     PlcTask Inputs/GVL_iXlinker.EtherCAT_Master_EJxxxx.Beckhoff_EJx9xx.A_0005_EJ1957_0000_0017.Module_1_FSOE.FSoE_Inputs.FSOE/FSIN_Module_4_Channel_2_Input <-> Module 1 (FSOE)/FSoE Inputs/FSOE/FSIN Module 4.Channel 2.Input
//     PlcTask Inputs/GVL_iXlinker.EtherCAT_Master_EJxxxx.Beckhoff_EJx9xx.A_0005_EJ1957_0000_0017.Module_1_FSOE.FSoE_Inputs.FSOE/FSIN_Module_1_Module_Fault <-> Module 1 (FSOE)/FSoE Inputs/FSOE/FSIN Module 1.Module Fault
//     PlcTask Inputs/GVL_iXlinker.EtherCAT_Master_EJxxxx.Beckhoff_EJx9xx.A_0005_EJ1957_0000_0017.Module_1_FSOE.FSoE_Inputs.FSOE/FSIN_Module_2_Module_Fault <-> Module 1 (FSOE)/FSoE Inputs/FSOE/FSIN Module 2.Module Fault
//     PlcTask Inputs/GVL_iXlinker.EtherCAT_Master_EJxxxx.Beckhoff_EJx9xx.A_0005_EJ1957_0000_0017.Module_1_FSOE.FSoE_Inputs.FSOE/FSIN_Module_3_Module_Fault <-> Module 1 (FSOE)/FSoE Inputs/FSOE/FSIN Module 3.Module Fault
//     PlcTask Inputs/GVL_iXlinker.EtherCAT_Master_EJxxxx.Beckhoff_EJx9xx.A_0005_EJ1957_0000_0017.Module_1_FSOE.FSoE_Inputs.FSOE/FSIN_Module_4_Module_Fault <-> Module 1 (FSOE)/FSoE Inputs/FSOE/FSIN Module 4.Module Fault
//     PlcTask Inputs/GVL_iXlinker.EtherCAT_Master_EJxxxx.Beckhoff_EJx9xx.A_0005_EJ1957_0000_0017.Module_1_FSOE.FSoE_Inputs.FSOE/FSoE_CRC_000 <-> Module 1 (FSOE)/FSoE Inputs/FSOE/FSoE CRC 000
//     PlcTask Inputs/GVL_iXlinker.EtherCAT_Master_EJxxxx.Beckhoff_EJx9xx.A_0005_EJ1957_0000_0017.Module_1_FSOE.FSoE_Inputs.FSOE/FSoE_Connection_ID <-> Module 1 (FSOE)/FSoE Inputs/FSOE/FSoE Connection ID
//     PlcTask Outputs/GVL_iXlinker.EtherCAT_Master_EJxxxx.Beckhoff_EJx9xx.A_0005_EJ1957_0000_0017.Module_1_FSOE.FSoE_Outputs.FSOE/FSoE_Command <-> Module 1 (FSOE)/FSoE Outputs/FSOE/FSoE Command
//     PlcTask Outputs/GVL_iXlinker.EtherCAT_Master_EJxxxx.Beckhoff_EJx9xx.A_0005_EJ1957_0000_0017.Module_1_FSOE.FSoE_Outputs.FSOE/FSOUT_Module_Channel_1_Output <-> Module 1 (FSOE)/FSoE Outputs/FSOE/FSOUT Module.Channel 1.Output
//     PlcTask Outputs/GVL_iXlinker.EtherCAT_Master_EJxxxx.Beckhoff_EJx9xx.A_0005_EJ1957_0000_0017.Module_1_FSOE.FSoE_Outputs.FSOE/FSOUT_Module_Channel_2_Output <-> Module 1 (FSOE)/FSoE Outputs/FSOE/FSOUT Module.Channel 2.Output
//     PlcTask Outputs/GVL_iXlinker.EtherCAT_Master_EJxxxx.Beckhoff_EJx9xx.A_0005_EJ1957_0000_0017.Module_1_FSOE.FSoE_Outputs.FSOE/FSOUT_Module_Channel_3_Output <-> Module 1 (FSOE)/FSoE Outputs/FSOE/FSOUT Module.Channel 3.Output
//     PlcTask Outputs/GVL_iXlinker.EtherCAT_Master_EJxxxx.Beckhoff_EJx9xx.A_0005_EJ1957_0000_0017.Module_1_FSOE.FSoE_Outputs.FSOE/FSOUT_Module_Channel_4_Output <-> Module 1 (FSOE)/FSoE Outputs/FSOE/FSOUT Module.Channel 4.Output
//     PlcTask Outputs/GVL_iXlinker.EtherCAT_Master_EJxxxx.Beckhoff_EJx9xx.A_0005_EJ1957_0000_0017.Module_1_FSOE.FSoE_Outputs.FSOE/FSOUT_Module_ErrAck <-> Module 1 (FSOE)/FSoE Outputs/FSOE/FSOUT Module.ErrAck
//     PlcTask Outputs/GVL_iXlinker.EtherCAT_Master_EJxxxx.Beckhoff_EJx9xx.A_0005_EJ1957_0000_0017.Module_1_FSOE.FSoE_Outputs.FSOE/FSIN_Module_1_ErrAck <-> Module 1 (FSOE)/FSoE Outputs/FSOE/FSIN Module 1.ErrAck
//     PlcTask Outputs/GVL_iXlinker.EtherCAT_Master_EJxxxx.Beckhoff_EJx9xx.A_0005_EJ1957_0000_0017.Module_1_FSOE.FSoE_Outputs.FSOE/FSIN_Module_2_ErrAck <-> Module 1 (FSOE)/FSoE Outputs/FSOE/FSIN Module 2.ErrAck
//     PlcTask Outputs/GVL_iXlinker.EtherCAT_Master_EJxxxx.Beckhoff_EJx9xx.A_0005_EJ1957_0000_0017.Module_1_FSOE.FSoE_Outputs.FSOE/FSIN_Module_3_ErrAck <-> Module 1 (FSOE)/FSoE Outputs/FSOE/FSIN Module 3.ErrAck
//     PlcTask Outputs/GVL_iXlinker.EtherCAT_Master_EJxxxx.Beckhoff_EJx9xx.A_0005_EJ1957_0000_0017.Module_1_FSOE.FSoE_Outputs.FSOE/FSIN_Module_4_ErrAck <-> Module 1 (FSOE)/FSoE Outputs/FSOE/FSIN Module 4.ErrAck
//     PlcTask Outputs/GVL_iXlinker.EtherCAT_Master_EJxxxx.Beckhoff_EJx9xx.A_0005_EJ1957_0000_0017.Module_1_FSOE.FSoE_Outputs.FSOE/FSoE_CRC_000 <-> Module 1 (FSOE)/FSoE Outputs/FSOE/FSoE CRC 000
//     PlcTask Outputs/GVL_iXlinker.EtherCAT_Master_EJxxxx.Beckhoff_EJx9xx.A_0005_EJ1957_0000_0017.Module_1_FSOE.FSoE_Outputs.FSOE/FSoE_Connection_ID <-> Module 1 (FSOE)/FSoE Outputs/FSOE/FSoE Connection ID
//     PlcTask Outputs/GVL_iXlinker.EtherCAT_Master_EJxxxx.Beckhoff_EJx9xx.A_0005_EJ1957_0000_0017.Module_2_FSOUT.Outputs.Channel_1_Standard_Output <-> Module 2 (FSOUT)/Outputs/Channel 1.Standard Output
//     PlcTask Outputs/GVL_iXlinker.EtherCAT_Master_EJxxxx.Beckhoff_EJx9xx.A_0005_EJ1957_0000_0017.Module_2_FSOUT.Outputs.Channel_2_Standard_Output <-> Module 2 (FSOUT)/Outputs/Channel 2.Standard Output
//     PlcTask Outputs/GVL_iXlinker.EtherCAT_Master_EJxxxx.Beckhoff_EJx9xx.A_0005_EJ1957_0000_0017.Module_2_FSOUT.Outputs.Channel_3_Standard_Output <-> Module 2 (FSOUT)/Outputs/Channel 3.Standard Output
//     PlcTask Outputs/GVL_iXlinker.EtherCAT_Master_EJxxxx.Beckhoff_EJx9xx.A_0005_EJ1957_0000_0017.Module_2_FSOUT.Outputs.Channel_4_Standard_Output <-> Module 2 (FSOUT)/Outputs/Channel 4.Standard Output
//     PlcTask Inputs/GVL_iXlinker.EtherCAT_Master_EJxxxx.Beckhoff_EJx9xx.A_0005_EJ1957_0000_0017.Module_3_DEVICEIO.FIELDVOLTAGE_Field_Voltage_Status.Fieldvoltage_Underrange <-> Module 3 (DEVICEIO)/FIELDVOLTAGE Field Voltage Status/Fieldvoltage Underrange
//     PlcTask Inputs/GVL_iXlinker.EtherCAT_Master_EJxxxx.Beckhoff_EJx9xx.A_0005_EJ1957_0000_0017.Module_3_DEVICEIO.FIELDVOLTAGE_Field_Voltage_Status.Fieldvoltage_Overrange <-> Module 3 (DEVICEIO)/FIELDVOLTAGE Field Voltage Status/Fieldvoltage Overrange
//     PlcTask Inputs/GVL_iXlinker.EtherCAT_Master_EJxxxx.Beckhoff_EJx9xx.A_0005_EJ1957_0000_0017.Module_4_FSLOGIC.FSLOGIC_Inputs.Safe_Logic_State <-> Module 4 (FSLOGIC)/FSLOGIC Inputs/Safe Logic State
//     PlcTask Inputs/GVL_iXlinker.EtherCAT_Master_EJxxxx.Beckhoff_EJx9xx.A_0005_EJ1957_0000_0017.Module_4_FSLOGIC.FSLOGIC_Inputs.Cycle_Counter <-> Module 4 (FSLOGIC)/FSLOGIC Inputs/Cycle Counter
//     PlcTask Inputs/GVL_iXlinker.EtherCAT_Master_EJxxxx.Beckhoff_EJx9xx.A_0005_EJ1957_0000_0017.WcState.WcState0 <-> WcState/WcState0
//     PlcTask Inputs/GVL_iXlinker.EtherCAT_Master_EJxxxx.Beckhoff_EJx9xx.A_0005_EJ1957_0000_0017.WcState.WcState1 <-> WcState/WcState1
//     PlcTask Inputs/GVL_iXlinker.EtherCAT_Master_EJxxxx.Beckhoff_EJx9xx.A_0005_EJ1957_0000_0017.WcState.InputToggle0 <-> WcState/InputToggle0
//     PlcTask Inputs/GVL_iXlinker.EtherCAT_Master_EJxxxx.Beckhoff_EJx9xx.A_0005_EJ1957_0000_0017.WcState.InputToggle1 <-> WcState/InputToggle1
//     PlcTask Inputs/GVL_iXlinker.EtherCAT_Master_EJxxxx.Beckhoff_EJx9xx.A_0005_EJ1957_0000_0017.InfoData.AdsAddr <-> InfoData/AdsAddr
//     PlcTask Inputs/GVL_iXlinker.EtherCAT_Master_EJxxxx.Beckhoff_EJx9xx.A_0005_EJ1957_0000_0017.InfoData.State <-> InfoData/State
//   PLC/PLC Instance <-> EtherCAT Master EJxxxx/Beckhoff EJx9xx/A_0006(EJ1957-0000-0018)
//     PlcTask Inputs/GVL_iXlinker.EtherCAT_Master_EJxxxx.Beckhoff_EJx9xx.A_0006_EJ1957_0000_0018.Module_1_FSOE.FSoE_Inputs.FSOE/FSoE_Command <-> Module 1 (FSOE)/FSoE Inputs/FSOE/FSoE Command
//     PlcTask Inputs/GVL_iXlinker.EtherCAT_Master_EJxxxx.Beckhoff_EJx9xx.A_0006_EJ1957_0000_0018.Module_1_FSOE.FSoE_Inputs.FSOE/FSOUT_Module_Module_Fault <-> Module 1 (FSOE)/FSoE Inputs/FSOE/FSOUT Module.Module Fault
//     PlcTask Inputs/GVL_iXlinker.EtherCAT_Master_EJxxxx.Beckhoff_EJx9xx.A_0006_EJ1957_0000_0018.Module_1_FSOE.FSoE_Inputs.FSOE/FSIN_Module_1_Channel_1_Input <-> Module 1 (FSOE)/FSoE Inputs/FSOE/FSIN Module 1.Channel 1.Input
//     PlcTask Inputs/GVL_iXlinker.EtherCAT_Master_EJxxxx.Beckhoff_EJx9xx.A_0006_EJ1957_0000_0018.Module_1_FSOE.FSoE_Inputs.FSOE/FSIN_Module_1_Channel_2_Input <-> Module 1 (FSOE)/FSoE Inputs/FSOE/FSIN Module 1.Channel 2.Input
//     PlcTask Inputs/GVL_iXlinker.EtherCAT_Master_EJxxxx.Beckhoff_EJx9xx.A_0006_EJ1957_0000_0018.Module_1_FSOE.FSoE_Inputs.FSOE/FSIN_Module_2_Channel_1_Input <-> Module 1 (FSOE)/FSoE Inputs/FSOE/FSIN Module 2.Channel 1.Input
//     PlcTask Inputs/GVL_iXlinker.EtherCAT_Master_EJxxxx.Beckhoff_EJx9xx.A_0006_EJ1957_0000_0018.Module_1_FSOE.FSoE_Inputs.FSOE/FSIN_Module_2_Channel_2_Input <-> Module 1 (FSOE)/FSoE Inputs/FSOE/FSIN Module 2.Channel 2.Input
//     PlcTask Inputs/GVL_iXlinker.EtherCAT_Master_EJxxxx.Beckhoff_EJx9xx.A_0006_EJ1957_0000_0018.Module_1_FSOE.FSoE_Inputs.FSOE/FSIN_Module_3_Channel_1_Input <-> Module 1 (FSOE)/FSoE Inputs/FSOE/FSIN Module 3.Channel 1.Input
//     PlcTask Inputs/GVL_iXlinker.EtherCAT_Master_EJxxxx.Beckhoff_EJx9xx.A_0006_EJ1957_0000_0018.Module_1_FSOE.FSoE_Inputs.FSOE/FSIN_Module_3_Channel_2_Input <-> Module 1 (FSOE)/FSoE Inputs/FSOE/FSIN Module 3.Channel 2.Input
//     PlcTask Inputs/GVL_iXlinker.EtherCAT_Master_EJxxxx.Beckhoff_EJx9xx.A_0006_EJ1957_0000_0018.Module_1_FSOE.FSoE_Inputs.FSOE/FSIN_Module_4_Channel_1_Input <-> Module 1 (FSOE)/FSoE Inputs/FSOE/FSIN Module 4.Channel 1.Input
//     PlcTask Inputs/GVL_iXlinker.EtherCAT_Master_EJxxxx.Beckhoff_EJx9xx.A_0006_EJ1957_0000_0018.Module_1_FSOE.FSoE_Inputs.FSOE/FSIN_Module_4_Channel_2_Input <-> Module 1 (FSOE)/FSoE Inputs/FSOE/FSIN Module 4.Channel 2.Input
//     PlcTask Inputs/GVL_iXlinker.EtherCAT_Master_EJxxxx.Beckhoff_EJx9xx.A_0006_EJ1957_0000_0018.Module_1_FSOE.FSoE_Inputs.FSOE/FSIN_Module_1_Module_Fault <-> Module 1 (FSOE)/FSoE Inputs/FSOE/FSIN Module 1.Module Fault
//     PlcTask Inputs/GVL_iXlinker.EtherCAT_Master_EJxxxx.Beckhoff_EJx9xx.A_0006_EJ1957_0000_0018.Module_1_FSOE.FSoE_Inputs.FSOE/FSIN_Module_2_Module_Fault <-> Module 1 (FSOE)/FSoE Inputs/FSOE/FSIN Module 2.Module Fault
//     PlcTask Inputs/GVL_iXlinker.EtherCAT_Master_EJxxxx.Beckhoff_EJx9xx.A_0006_EJ1957_0000_0018.Module_1_FSOE.FSoE_Inputs.FSOE/FSIN_Module_3_Module_Fault <-> Module 1 (FSOE)/FSoE Inputs/FSOE/FSIN Module 3.Module Fault
//     PlcTask Inputs/GVL_iXlinker.EtherCAT_Master_EJxxxx.Beckhoff_EJx9xx.A_0006_EJ1957_0000_0018.Module_1_FSOE.FSoE_Inputs.FSOE/FSIN_Module_4_Module_Fault <-> Module 1 (FSOE)/FSoE Inputs/FSOE/FSIN Module 4.Module Fault
//     PlcTask Inputs/GVL_iXlinker.EtherCAT_Master_EJxxxx.Beckhoff_EJx9xx.A_0006_EJ1957_0000_0018.Module_1_FSOE.FSoE_Inputs.FSOE/FSoE_CRC_000 <-> Module 1 (FSOE)/FSoE Inputs/FSOE/FSoE CRC 000
//     PlcTask Inputs/GVL_iXlinker.EtherCAT_Master_EJxxxx.Beckhoff_EJx9xx.A_0006_EJ1957_0000_0018.Module_1_FSOE.FSoE_Inputs.FSOE/FSoE_Connection_ID <-> Module 1 (FSOE)/FSoE Inputs/FSOE/FSoE Connection ID
//     PlcTask Outputs/GVL_iXlinker.EtherCAT_Master_EJxxxx.Beckhoff_EJx9xx.A_0006_EJ1957_0000_0018.Module_1_FSOE.FSoE_Outputs.FSOE/FSoE_Command <-> Module 1 (FSOE)/FSoE Outputs/FSOE/FSoE Command
//     PlcTask Outputs/GVL_iXlinker.EtherCAT_Master_EJxxxx.Beckhoff_EJx9xx.A_0006_EJ1957_0000_0018.Module_1_FSOE.FSoE_Outputs.FSOE/FSOUT_Module_Channel_1_Output <-> Module 1 (FSOE)/FSoE Outputs/FSOE/FSOUT Module.Channel 1.Output
//     PlcTask Outputs/GVL_iXlinker.EtherCAT_Master_EJxxxx.Beckhoff_EJx9xx.A_0006_EJ1957_0000_0018.Module_1_FSOE.FSoE_Outputs.FSOE/FSOUT_Module_Channel_2_Output <-> Module 1 (FSOE)/FSoE Outputs/FSOE/FSOUT Module.Channel 2.Output
//     PlcTask Outputs/GVL_iXlinker.EtherCAT_Master_EJxxxx.Beckhoff_EJx9xx.A_0006_EJ1957_0000_0018.Module_1_FSOE.FSoE_Outputs.FSOE/FSOUT_Module_Channel_3_Output <-> Module 1 (FSOE)/FSoE Outputs/FSOE/FSOUT Module.Channel 3.Output
//     PlcTask Outputs/GVL_iXlinker.EtherCAT_Master_EJxxxx.Beckhoff_EJx9xx.A_0006_EJ1957_0000_0018.Module_1_FSOE.FSoE_Outputs.FSOE/FSOUT_Module_Channel_4_Output <-> Module 1 (FSOE)/FSoE Outputs/FSOE/FSOUT Module.Channel 4.Output
//     PlcTask Outputs/GVL_iXlinker.EtherCAT_Master_EJxxxx.Beckhoff_EJx9xx.A_0006_EJ1957_0000_0018.Module_1_FSOE.FSoE_Outputs.FSOE/FSOUT_Module_ErrAck <-> Module 1 (FSOE)/FSoE Outputs/FSOE/FSOUT Module.ErrAck
//     PlcTask Outputs/GVL_iXlinker.EtherCAT_Master_EJxxxx.Beckhoff_EJx9xx.A_0006_EJ1957_0000_0018.Module_1_FSOE.FSoE_Outputs.FSOE/FSIN_Module_1_ErrAck <-> Module 1 (FSOE)/FSoE Outputs/FSOE/FSIN Module 1.ErrAck
//     PlcTask Outputs/GVL_iXlinker.EtherCAT_Master_EJxxxx.Beckhoff_EJx9xx.A_0006_EJ1957_0000_0018.Module_1_FSOE.FSoE_Outputs.FSOE/FSIN_Module_2_ErrAck <-> Module 1 (FSOE)/FSoE Outputs/FSOE/FSIN Module 2.ErrAck
//     PlcTask Outputs/GVL_iXlinker.EtherCAT_Master_EJxxxx.Beckhoff_EJx9xx.A_0006_EJ1957_0000_0018.Module_1_FSOE.FSoE_Outputs.FSOE/FSIN_Module_3_ErrAck <-> Module 1 (FSOE)/FSoE Outputs/FSOE/FSIN Module 3.ErrAck
//     PlcTask Outputs/GVL_iXlinker.EtherCAT_Master_EJxxxx.Beckhoff_EJx9xx.A_0006_EJ1957_0000_0018.Module_1_FSOE.FSoE_Outputs.FSOE/FSIN_Module_4_ErrAck <-> Module 1 (FSOE)/FSoE Outputs/FSOE/FSIN Module 4.ErrAck
//     PlcTask Outputs/GVL_iXlinker.EtherCAT_Master_EJxxxx.Beckhoff_EJx9xx.A_0006_EJ1957_0000_0018.Module_1_FSOE.FSoE_Outputs.FSOE/FSoE_CRC_000 <-> Module 1 (FSOE)/FSoE Outputs/FSOE/FSoE CRC 000
//     PlcTask Outputs/GVL_iXlinker.EtherCAT_Master_EJxxxx.Beckhoff_EJx9xx.A_0006_EJ1957_0000_0018.Module_1_FSOE.FSoE_Outputs.FSOE/FSoE_Connection_ID <-> Module 1 (FSOE)/FSoE Outputs/FSOE/FSoE Connection ID
//     PlcTask Outputs/GVL_iXlinker.EtherCAT_Master_EJxxxx.Beckhoff_EJx9xx.A_0006_EJ1957_0000_0018.Module_2_FSOUT.Outputs.Channel_1_Standard_Output <-> Module 2 (FSOUT)/Outputs/Channel 1.Standard Output
//     PlcTask Outputs/GVL_iXlinker.EtherCAT_Master_EJxxxx.Beckhoff_EJx9xx.A_0006_EJ1957_0000_0018.Module_2_FSOUT.Outputs.Channel_2_Standard_Output <-> Module 2 (FSOUT)/Outputs/Channel 2.Standard Output
//     PlcTask Outputs/GVL_iXlinker.EtherCAT_Master_EJxxxx.Beckhoff_EJx9xx.A_0006_EJ1957_0000_0018.Module_2_FSOUT.Outputs.Channel_3_Standard_Output <-> Module 2 (FSOUT)/Outputs/Channel 3.Standard Output
//     PlcTask Outputs/GVL_iXlinker.EtherCAT_Master_EJxxxx.Beckhoff_EJx9xx.A_0006_EJ1957_0000_0018.Module_2_FSOUT.Outputs.Channel_4_Standard_Output <-> Module 2 (FSOUT)/Outputs/Channel 4.Standard Output
//     PlcTask Inputs/GVL_iXlinker.EtherCAT_Master_EJxxxx.Beckhoff_EJx9xx.A_0006_EJ1957_0000_0018.Module_3_DEVICEIO.FIELDVOLTAGE_Field_Voltage_Status.Fieldvoltage_Underrange <-> Module 3 (DEVICEIO)/FIELDVOLTAGE Field Voltage Status/Fieldvoltage Underrange
//     PlcTask Inputs/GVL_iXlinker.EtherCAT_Master_EJxxxx.Beckhoff_EJx9xx.A_0006_EJ1957_0000_0018.Module_3_DEVICEIO.FIELDVOLTAGE_Field_Voltage_Status.Fieldvoltage_Overrange <-> Module 3 (DEVICEIO)/FIELDVOLTAGE Field Voltage Status/Fieldvoltage Overrange
//     PlcTask Inputs/GVL_iXlinker.EtherCAT_Master_EJxxxx.Beckhoff_EJx9xx.A_0006_EJ1957_0000_0018.Module_4_FSLOGIC.FSLOGIC_Inputs.Safe_Logic_State <-> Module 4 (FSLOGIC)/FSLOGIC Inputs/Safe Logic State
//     PlcTask Inputs/GVL_iXlinker.EtherCAT_Master_EJxxxx.Beckhoff_EJx9xx.A_0006_EJ1957_0000_0018.Module_4_FSLOGIC.FSLOGIC_Inputs.Cycle_Counter <-> Module 4 (FSLOGIC)/FSLOGIC Inputs/Cycle Counter
//     PlcTask Inputs/GVL_iXlinker.EtherCAT_Master_EJxxxx.Beckhoff_EJx9xx.A_0006_EJ1957_0000_0018.WcState.WcState0 <-> WcState/WcState0
//     PlcTask Inputs/GVL_iXlinker.EtherCAT_Master_EJxxxx.Beckhoff_EJx9xx.A_0006_EJ1957_0000_0018.WcState.WcState1 <-> WcState/WcState1
//     PlcTask Inputs/GVL_iXlinker.EtherCAT_Master_EJxxxx.Beckhoff_EJx9xx.A_0006_EJ1957_0000_0018.WcState.InputToggle0 <-> WcState/InputToggle0
//     PlcTask Inputs/GVL_iXlinker.EtherCAT_Master_EJxxxx.Beckhoff_EJx9xx.A_0006_EJ1957_0000_0018.WcState.InputToggle1 <-> WcState/InputToggle1
//     PlcTask Inputs/GVL_iXlinker.EtherCAT_Master_EJxxxx.Beckhoff_EJx9xx.A_0006_EJ1957_0000_0018.InfoData.AdsAddr <-> InfoData/AdsAddr
//     PlcTask Inputs/GVL_iXlinker.EtherCAT_Master_EJxxxx.Beckhoff_EJx9xx.A_0006_EJ1957_0000_0018.InfoData.State <-> InfoData/State
//   PLC/PLC Instance <-> EtherCAT Master EJxxxx/Beckhoff EJx9xx/A_0007(EJ2914-0000-0017)
//     PlcTask Inputs/GVL_iXlinker.EtherCAT_Master_EJxxxx.Beckhoff_EJx9xx.A_0007_EJ2914_0000_0017.Module_1_FSOE.FSoE_Inputs.FSOE/FSoE_Command <-> Module 1 (FSOE)/FSoE Inputs/FSOE/FSoE Command
//     PlcTask Inputs/GVL_iXlinker.EtherCAT_Master_EJxxxx.Beckhoff_EJx9xx.A_0007_EJ2914_0000_0017.Module_1_FSOE.FSoE_Inputs.FSOE/FSOUT_Module_Module_Fault <-> Module 1 (FSOE)/FSoE Inputs/FSOE/FSOUT Module.Module Fault
//     PlcTask Inputs/GVL_iXlinker.EtherCAT_Master_EJxxxx.Beckhoff_EJx9xx.A_0007_EJ2914_0000_0017.Module_1_FSOE.FSoE_Inputs.FSOE/FSoE_CRC_000 <-> Module 1 (FSOE)/FSoE Inputs/FSOE/FSoE CRC 000
//     PlcTask Inputs/GVL_iXlinker.EtherCAT_Master_EJxxxx.Beckhoff_EJx9xx.A_0007_EJ2914_0000_0017.Module_1_FSOE.FSoE_Inputs.FSOE/FSoE_Connection_ID <-> Module 1 (FSOE)/FSoE Inputs/FSOE/FSoE Connection ID
//     PlcTask Outputs/GVL_iXlinker.EtherCAT_Master_EJxxxx.Beckhoff_EJx9xx.A_0007_EJ2914_0000_0017.Module_1_FSOE.FSoE_Outputs.FSOE/FSoE_Command <-> Module 1 (FSOE)/FSoE Outputs/FSOE/FSoE Command
//     PlcTask Outputs/GVL_iXlinker.EtherCAT_Master_EJxxxx.Beckhoff_EJx9xx.A_0007_EJ2914_0000_0017.Module_1_FSOE.FSoE_Outputs.FSOE/FSOUT_Module_Channel_1_Output <-> Module 1 (FSOE)/FSoE Outputs/FSOE/FSOUT Module.Channel 1.Output
//     PlcTask Outputs/GVL_iXlinker.EtherCAT_Master_EJxxxx.Beckhoff_EJx9xx.A_0007_EJ2914_0000_0017.Module_1_FSOE.FSoE_Outputs.FSOE/FSOUT_Module_Channel_2_Output <-> Module 1 (FSOE)/FSoE Outputs/FSOE/FSOUT Module.Channel 2.Output
//     PlcTask Outputs/GVL_iXlinker.EtherCAT_Master_EJxxxx.Beckhoff_EJx9xx.A_0007_EJ2914_0000_0017.Module_1_FSOE.FSoE_Outputs.FSOE/FSOUT_Module_Channel_3_Output <-> Module 1 (FSOE)/FSoE Outputs/FSOE/FSOUT Module.Channel 3.Output
//     PlcTask Outputs/GVL_iXlinker.EtherCAT_Master_EJxxxx.Beckhoff_EJx9xx.A_0007_EJ2914_0000_0017.Module_1_FSOE.FSoE_Outputs.FSOE/FSOUT_Module_Channel_4_Output <-> Module 1 (FSOE)/FSoE Outputs/FSOE/FSOUT Module.Channel 4.Output
//     PlcTask Outputs/GVL_iXlinker.EtherCAT_Master_EJxxxx.Beckhoff_EJx9xx.A_0007_EJ2914_0000_0017.Module_1_FSOE.FSoE_Outputs.FSOE/FSOUT_Module_ErrAck <-> Module 1 (FSOE)/FSoE Outputs/FSOE/FSOUT Module.ErrAck
//     PlcTask Outputs/GVL_iXlinker.EtherCAT_Master_EJxxxx.Beckhoff_EJx9xx.A_0007_EJ2914_0000_0017.Module_1_FSOE.FSoE_Outputs.FSOE/FSoE_CRC_000 <-> Module 1 (FSOE)/FSoE Outputs/FSOE/FSoE CRC 000
//     PlcTask Outputs/GVL_iXlinker.EtherCAT_Master_EJxxxx.Beckhoff_EJx9xx.A_0007_EJ2914_0000_0017.Module_1_FSOE.FSoE_Outputs.FSOE/FSoE_Connection_ID <-> Module 1 (FSOE)/FSoE Outputs/FSOE/FSoE Connection ID
//     PlcTask Outputs/GVL_iXlinker.EtherCAT_Master_EJxxxx.Beckhoff_EJx9xx.A_0007_EJ2914_0000_0017.Module_2_FSOUT.Outputs.Channel_1_Standard_Output <-> Module 2 (FSOUT)/Outputs/Channel 1.Standard Output
//     PlcTask Outputs/GVL_iXlinker.EtherCAT_Master_EJxxxx.Beckhoff_EJx9xx.A_0007_EJ2914_0000_0017.Module_2_FSOUT.Outputs.Channel_2_Standard_Output <-> Module 2 (FSOUT)/Outputs/Channel 2.Standard Output
//     PlcTask Outputs/GVL_iXlinker.EtherCAT_Master_EJxxxx.Beckhoff_EJx9xx.A_0007_EJ2914_0000_0017.Module_2_FSOUT.Outputs.Channel_3_Standard_Output <-> Module 2 (FSOUT)/Outputs/Channel 3.Standard Output
//     PlcTask Outputs/GVL_iXlinker.EtherCAT_Master_EJxxxx.Beckhoff_EJx9xx.A_0007_EJ2914_0000_0017.Module_2_FSOUT.Outputs.Channel_4_Standard_Output <-> Module 2 (FSOUT)/Outputs/Channel 4.Standard Output
//     PlcTask Inputs/GVL_iXlinker.EtherCAT_Master_EJxxxx.Beckhoff_EJx9xx.A_0007_EJ2914_0000_0017.Module_3_DEVICEIO.FIELDVOLTAGE_Field_Voltage_Status.Fieldvoltage_Underrange <-> Module 3 (DEVICEIO)/FIELDVOLTAGE Field Voltage Status/Fieldvoltage Underrange
//     PlcTask Inputs/GVL_iXlinker.EtherCAT_Master_EJxxxx.Beckhoff_EJx9xx.A_0007_EJ2914_0000_0017.Module_3_DEVICEIO.FIELDVOLTAGE_Field_Voltage_Status.Fieldvoltage_Overrange <-> Module 3 (DEVICEIO)/FIELDVOLTAGE Field Voltage Status/Fieldvoltage Overrange
//     PlcTask Inputs/GVL_iXlinker.EtherCAT_Master_EJxxxx.Beckhoff_EJx9xx.A_0007_EJ2914_0000_0017.Module_4_FSLOGIC.FSLOGIC_Inputs.Safe_Logic_State <-> Module 4 (FSLOGIC)/FSLOGIC Inputs/Safe Logic State
//     PlcTask Inputs/GVL_iXlinker.EtherCAT_Master_EJxxxx.Beckhoff_EJx9xx.A_0007_EJ2914_0000_0017.Module_4_FSLOGIC.FSLOGIC_Inputs.Cycle_Counter <-> Module 4 (FSLOGIC)/FSLOGIC Inputs/Cycle Counter
//     PlcTask Inputs/GVL_iXlinker.EtherCAT_Master_EJxxxx.Beckhoff_EJx9xx.A_0007_EJ2914_0000_0017.WcState.WcState0 <-> WcState/WcState0
//     PlcTask Inputs/GVL_iXlinker.EtherCAT_Master_EJxxxx.Beckhoff_EJx9xx.A_0007_EJ2914_0000_0017.WcState.WcState1 <-> WcState/WcState1
//     PlcTask Inputs/GVL_iXlinker.EtherCAT_Master_EJxxxx.Beckhoff_EJx9xx.A_0007_EJ2914_0000_0017.WcState.InputToggle0 <-> WcState/InputToggle0
//     PlcTask Inputs/GVL_iXlinker.EtherCAT_Master_EJxxxx.Beckhoff_EJx9xx.A_0007_EJ2914_0000_0017.WcState.InputToggle1 <-> WcState/InputToggle1
//     PlcTask Inputs/GVL_iXlinker.EtherCAT_Master_EJxxxx.Beckhoff_EJx9xx.A_0007_EJ2914_0000_0017.InfoData.AdsAddr <-> InfoData/AdsAddr
//     PlcTask Inputs/GVL_iXlinker.EtherCAT_Master_EJxxxx.Beckhoff_EJx9xx.A_0007_EJ2914_0000_0017.InfoData.State <-> InfoData/State
//   PLC/PLC Instance <-> EtherCAT Master EJxxxx/Beckhoff EJx9xx/A_0008(EJ2914-0000-0018)
//     PlcTask Inputs/GVL_iXlinker.EtherCAT_Master_EJxxxx.Beckhoff_EJx9xx.A_0008_EJ2914_0000_0018.Module_1_FSOE.FSoE_Inputs.FSOE/FSoE_Command <-> Module 1 (FSOE)/FSoE Inputs/FSOE/FSoE Command
//     PlcTask Inputs/GVL_iXlinker.EtherCAT_Master_EJxxxx.Beckhoff_EJx9xx.A_0008_EJ2914_0000_0018.Module_1_FSOE.FSoE_Inputs.FSOE/FSOUT_Module_Module_Fault <-> Module 1 (FSOE)/FSoE Inputs/FSOE/FSOUT Module.Module Fault
//     PlcTask Inputs/GVL_iXlinker.EtherCAT_Master_EJxxxx.Beckhoff_EJx9xx.A_0008_EJ2914_0000_0018.Module_1_FSOE.FSoE_Inputs.FSOE/FSoE_CRC_000 <-> Module 1 (FSOE)/FSoE Inputs/FSOE/FSoE CRC 000
//     PlcTask Inputs/GVL_iXlinker.EtherCAT_Master_EJxxxx.Beckhoff_EJx9xx.A_0008_EJ2914_0000_0018.Module_1_FSOE.FSoE_Inputs.FSOE/FSoE_Connection_ID <-> Module 1 (FSOE)/FSoE Inputs/FSOE/FSoE Connection ID
//     PlcTask Outputs/GVL_iXlinker.EtherCAT_Master_EJxxxx.Beckhoff_EJx9xx.A_0008_EJ2914_0000_0018.Module_1_FSOE.FSoE_Outputs.FSOE/FSoE_Command <-> Module 1 (FSOE)/FSoE Outputs/FSOE/FSoE Command
//     PlcTask Outputs/GVL_iXlinker.EtherCAT_Master_EJxxxx.Beckhoff_EJx9xx.A_0008_EJ2914_0000_0018.Module_1_FSOE.FSoE_Outputs.FSOE/FSOUT_Module_Channel_1_Output <-> Module 1 (FSOE)/FSoE Outputs/FSOE/FSOUT Module.Channel 1.Output
//     PlcTask Outputs/GVL_iXlinker.EtherCAT_Master_EJxxxx.Beckhoff_EJx9xx.A_0008_EJ2914_0000_0018.Module_1_FSOE.FSoE_Outputs.FSOE/FSOUT_Module_Channel_2_Output <-> Module 1 (FSOE)/FSoE Outputs/FSOE/FSOUT Module.Channel 2.Output
//     PlcTask Outputs/GVL_iXlinker.EtherCAT_Master_EJxxxx.Beckhoff_EJx9xx.A_0008_EJ2914_0000_0018.Module_1_FSOE.FSoE_Outputs.FSOE/FSOUT_Module_Channel_3_Output <-> Module 1 (FSOE)/FSoE Outputs/FSOE/FSOUT Module.Channel 3.Output
//     PlcTask Outputs/GVL_iXlinker.EtherCAT_Master_EJxxxx.Beckhoff_EJx9xx.A_0008_EJ2914_0000_0018.Module_1_FSOE.FSoE_Outputs.FSOE/FSOUT_Module_Channel_4_Output <-> Module 1 (FSOE)/FSoE Outputs/FSOE/FSOUT Module.Channel 4.Output
//     PlcTask Outputs/GVL_iXlinker.EtherCAT_Master_EJxxxx.Beckhoff_EJx9xx.A_0008_EJ2914_0000_0018.Module_1_FSOE.FSoE_Outputs.FSOE/FSOUT_Module_ErrAck <-> Module 1 (FSOE)/FSoE Outputs/FSOE/FSOUT Module.ErrAck
//     PlcTask Outputs/GVL_iXlinker.EtherCAT_Master_EJxxxx.Beckhoff_EJx9xx.A_0008_EJ2914_0000_0018.Module_1_FSOE.FSoE_Outputs.FSOE/FSoE_CRC_000 <-> Module 1 (FSOE)/FSoE Outputs/FSOE/FSoE CRC 000
//     PlcTask Outputs/GVL_iXlinker.EtherCAT_Master_EJxxxx.Beckhoff_EJx9xx.A_0008_EJ2914_0000_0018.Module_1_FSOE.FSoE_Outputs.FSOE/FSoE_Connection_ID <-> Module 1 (FSOE)/FSoE Outputs/FSOE/FSoE Connection ID
//     PlcTask Outputs/GVL_iXlinker.EtherCAT_Master_EJxxxx.Beckhoff_EJx9xx.A_0008_EJ2914_0000_0018.Module_2_FSOUT.Outputs.Channel_1_Standard_Output <-> Module 2 (FSOUT)/Outputs/Channel 1.Standard Output
//     PlcTask Outputs/GVL_iXlinker.EtherCAT_Master_EJxxxx.Beckhoff_EJx9xx.A_0008_EJ2914_0000_0018.Module_2_FSOUT.Outputs.Channel_2_Standard_Output <-> Module 2 (FSOUT)/Outputs/Channel 2.Standard Output
//     PlcTask Outputs/GVL_iXlinker.EtherCAT_Master_EJxxxx.Beckhoff_EJx9xx.A_0008_EJ2914_0000_0018.Module_2_FSOUT.Outputs.Channel_3_Standard_Output <-> Module 2 (FSOUT)/Outputs/Channel 3.Standard Output
//     PlcTask Outputs/GVL_iXlinker.EtherCAT_Master_EJxxxx.Beckhoff_EJx9xx.A_0008_EJ2914_0000_0018.Module_2_FSOUT.Outputs.Channel_4_Standard_Output <-> Module 2 (FSOUT)/Outputs/Channel 4.Standard Output
//     PlcTask Inputs/GVL_iXlinker.EtherCAT_Master_EJxxxx.Beckhoff_EJx9xx.A_0008_EJ2914_0000_0018.Module_3_DEVICEIO.FIELDVOLTAGE_Field_Voltage_Status.Fieldvoltage_Underrange <-> Module 3 (DEVICEIO)/FIELDVOLTAGE Field Voltage Status/Fieldvoltage Underrange
//     PlcTask Inputs/GVL_iXlinker.EtherCAT_Master_EJxxxx.Beckhoff_EJx9xx.A_0008_EJ2914_0000_0018.Module_3_DEVICEIO.FIELDVOLTAGE_Field_Voltage_Status.Fieldvoltage_Overrange <-> Module 3 (DEVICEIO)/FIELDVOLTAGE Field Voltage Status/Fieldvoltage Overrange
//     PlcTask Inputs/GVL_iXlinker.EtherCAT_Master_EJxxxx.Beckhoff_EJx9xx.A_0008_EJ2914_0000_0018.Module_4_FSLOGIC.FSLOGIC_Inputs.Safe_Logic_State <-> Module 4 (FSLOGIC)/FSLOGIC Inputs/Safe Logic State
//     PlcTask Inputs/GVL_iXlinker.EtherCAT_Master_EJxxxx.Beckhoff_EJx9xx.A_0008_EJ2914_0000_0018.Module_4_FSLOGIC.FSLOGIC_Inputs.Cycle_Counter <-> Module 4 (FSLOGIC)/FSLOGIC Inputs/Cycle Counter
//     PlcTask Inputs/GVL_iXlinker.EtherCAT_Master_EJxxxx.Beckhoff_EJx9xx.A_0008_EJ2914_0000_0018.WcState.WcState0 <-> WcState/WcState0
//     PlcTask Inputs/GVL_iXlinker.EtherCAT_Master_EJxxxx.Beckhoff_EJx9xx.A_0008_EJ2914_0000_0018.WcState.WcState1 <-> WcState/WcState1
//     PlcTask Inputs/GVL_iXlinker.EtherCAT_Master_EJxxxx.Beckhoff_EJx9xx.A_0008_EJ2914_0000_0018.WcState.InputToggle0 <-> WcState/InputToggle0
//     PlcTask Inputs/GVL_iXlinker.EtherCAT_Master_EJxxxx.Beckhoff_EJx9xx.A_0008_EJ2914_0000_0018.WcState.InputToggle1 <-> WcState/InputToggle1
//     PlcTask Inputs/GVL_iXlinker.EtherCAT_Master_EJxxxx.Beckhoff_EJx9xx.A_0008_EJ2914_0000_0018.InfoData.AdsAddr <-> InfoData/AdsAddr
//     PlcTask Inputs/GVL_iXlinker.EtherCAT_Master_EJxxxx.Beckhoff_EJx9xx.A_0008_EJ2914_0000_0018.InfoData.State <-> InfoData/State
//   PLC/PLC Instance <-> EtherCAT Master EJxxxx/Beckhoff EJx9xx/A_0009(EJ2918-0000-0017)
//     PlcTask Inputs/GVL_iXlinker.EtherCAT_Master_EJxxxx.Beckhoff_EJx9xx.A_0009_EJ2918_0000_0017.Module_1_FSOE.FSoE_Inputs.FSOE/FSoE_Command <-> Module 1 (FSOE)/FSoE Inputs/FSOE/FSoE Command
//     PlcTask Inputs/GVL_iXlinker.EtherCAT_Master_EJxxxx.Beckhoff_EJx9xx.A_0009_EJ2918_0000_0017.Module_1_FSOE.FSoE_Inputs.FSOE/FSOUT_Module_1_Module_Fault <-> Module 1 (FSOE)/FSoE Inputs/FSOE/FSOUT Module 1.Module Fault
//     PlcTask Inputs/GVL_iXlinker.EtherCAT_Master_EJxxxx.Beckhoff_EJx9xx.A_0009_EJ2918_0000_0017.Module_1_FSOE.FSoE_Inputs.FSOE/FSOUT_Module_2_Module_Fault <-> Module 1 (FSOE)/FSoE Inputs/FSOE/FSOUT Module 2.Module Fault
//     PlcTask Inputs/GVL_iXlinker.EtherCAT_Master_EJxxxx.Beckhoff_EJx9xx.A_0009_EJ2918_0000_0017.Module_1_FSOE.FSoE_Inputs.FSOE/FSoE_CRC_000 <-> Module 1 (FSOE)/FSoE Inputs/FSOE/FSoE CRC 000
//     PlcTask Inputs/GVL_iXlinker.EtherCAT_Master_EJxxxx.Beckhoff_EJx9xx.A_0009_EJ2918_0000_0017.Module_1_FSOE.FSoE_Inputs.FSOE/FSoE_Connection_ID <-> Module 1 (FSOE)/FSoE Inputs/FSOE/FSoE Connection ID
//     PlcTask Outputs/GVL_iXlinker.EtherCAT_Master_EJxxxx.Beckhoff_EJx9xx.A_0009_EJ2918_0000_0017.Module_1_FSOE.FSoE_Outputs.FSOE/FSoE_Command <-> Module 1 (FSOE)/FSoE Outputs/FSOE/FSoE Command
//     PlcTask Outputs/GVL_iXlinker.EtherCAT_Master_EJxxxx.Beckhoff_EJx9xx.A_0009_EJ2918_0000_0017.Module_1_FSOE.FSoE_Outputs.FSOE/FSOUT_Module_1_Channel_1_Output <-> Module 1 (FSOE)/FSoE Outputs/FSOE/FSOUT Module 1.Channel 1.Output
//     PlcTask Outputs/GVL_iXlinker.EtherCAT_Master_EJxxxx.Beckhoff_EJx9xx.A_0009_EJ2918_0000_0017.Module_1_FSOE.FSoE_Outputs.FSOE/FSOUT_Module_1_Channel_2_Output <-> Module 1 (FSOE)/FSoE Outputs/FSOE/FSOUT Module 1.Channel 2.Output
//     PlcTask Outputs/GVL_iXlinker.EtherCAT_Master_EJxxxx.Beckhoff_EJx9xx.A_0009_EJ2918_0000_0017.Module_1_FSOE.FSoE_Outputs.FSOE/FSOUT_Module_1_Channel_3_Output <-> Module 1 (FSOE)/FSoE Outputs/FSOE/FSOUT Module 1.Channel 3.Output
//     PlcTask Outputs/GVL_iXlinker.EtherCAT_Master_EJxxxx.Beckhoff_EJx9xx.A_0009_EJ2918_0000_0017.Module_1_FSOE.FSoE_Outputs.FSOE/FSOUT_Module_1_Channel_4_Output <-> Module 1 (FSOE)/FSoE Outputs/FSOE/FSOUT Module 1.Channel 4.Output
//     PlcTask Outputs/GVL_iXlinker.EtherCAT_Master_EJxxxx.Beckhoff_EJx9xx.A_0009_EJ2918_0000_0017.Module_1_FSOE.FSoE_Outputs.FSOE/FSOUT_Module_2_Channel_1_Output <-> Module 1 (FSOE)/FSoE Outputs/FSOE/FSOUT Module 2.Channel 1.Output
//     PlcTask Outputs/GVL_iXlinker.EtherCAT_Master_EJxxxx.Beckhoff_EJx9xx.A_0009_EJ2918_0000_0017.Module_1_FSOE.FSoE_Outputs.FSOE/FSOUT_Module_2_Channel_2_Output <-> Module 1 (FSOE)/FSoE Outputs/FSOE/FSOUT Module 2.Channel 2.Output
//     PlcTask Outputs/GVL_iXlinker.EtherCAT_Master_EJxxxx.Beckhoff_EJx9xx.A_0009_EJ2918_0000_0017.Module_1_FSOE.FSoE_Outputs.FSOE/FSOUT_Module_2_Channel_3_Output <-> Module 1 (FSOE)/FSoE Outputs/FSOE/FSOUT Module 2.Channel 3.Output
//     PlcTask Outputs/GVL_iXlinker.EtherCAT_Master_EJxxxx.Beckhoff_EJx9xx.A_0009_EJ2918_0000_0017.Module_1_FSOE.FSoE_Outputs.FSOE/FSOUT_Module_2_Channel_4_Output <-> Module 1 (FSOE)/FSoE Outputs/FSOE/FSOUT Module 2.Channel 4.Output
//     PlcTask Outputs/GVL_iXlinker.EtherCAT_Master_EJxxxx.Beckhoff_EJx9xx.A_0009_EJ2918_0000_0017.Module_1_FSOE.FSoE_Outputs.FSOE/FSOUT_Module_1_ErrAck <-> Module 1 (FSOE)/FSoE Outputs/FSOE/FSOUT Module 1.ErrAck
//     PlcTask Outputs/GVL_iXlinker.EtherCAT_Master_EJxxxx.Beckhoff_EJx9xx.A_0009_EJ2918_0000_0017.Module_1_FSOE.FSoE_Outputs.FSOE/FSOUT_Module_2_ErrAck <-> Module 1 (FSOE)/FSoE Outputs/FSOE/FSOUT Module 2.ErrAck
//     PlcTask Outputs/GVL_iXlinker.EtherCAT_Master_EJxxxx.Beckhoff_EJx9xx.A_0009_EJ2918_0000_0017.Module_1_FSOE.FSoE_Outputs.FSOE/FSoE_CRC_000 <-> Module 1 (FSOE)/FSoE Outputs/FSOE/FSoE CRC 000
//     PlcTask Outputs/GVL_iXlinker.EtherCAT_Master_EJxxxx.Beckhoff_EJx9xx.A_0009_EJ2918_0000_0017.Module_1_FSOE.FSoE_Outputs.FSOE/FSoE_Connection_ID <-> Module 1 (FSOE)/FSoE Outputs/FSOE/FSoE Connection ID
//     PlcTask Outputs/GVL_iXlinker.EtherCAT_Master_EJxxxx.Beckhoff_EJx9xx.A_0009_EJ2918_0000_0017.Module_2_FSOUT.Outputs.Module_1_Channel_1_Standard_Output <-> Module 2 (FSOUT)/Outputs/Module 1.Channel 1.Standard Output
//     PlcTask Outputs/GVL_iXlinker.EtherCAT_Master_EJxxxx.Beckhoff_EJx9xx.A_0009_EJ2918_0000_0017.Module_2_FSOUT.Outputs.Module_1_Channel_2_Standard_Output <-> Module 2 (FSOUT)/Outputs/Module 1.Channel 2.Standard Output
//     PlcTask Outputs/GVL_iXlinker.EtherCAT_Master_EJxxxx.Beckhoff_EJx9xx.A_0009_EJ2918_0000_0017.Module_2_FSOUT.Outputs.Module_1_Channel_3_Standard_Output <-> Module 2 (FSOUT)/Outputs/Module 1.Channel 3.Standard Output
//     PlcTask Outputs/GVL_iXlinker.EtherCAT_Master_EJxxxx.Beckhoff_EJx9xx.A_0009_EJ2918_0000_0017.Module_2_FSOUT.Outputs.Module_1_Channel_4_Standard_Output <-> Module 2 (FSOUT)/Outputs/Module 1.Channel 4.Standard Output
//     PlcTask Outputs/GVL_iXlinker.EtherCAT_Master_EJxxxx.Beckhoff_EJx9xx.A_0009_EJ2918_0000_0017.Module_2_FSOUT.Outputs.Module_2_Channel_1_Standard_Output <-> Module 2 (FSOUT)/Outputs/Module 2.Channel 1.Standard Output
//     PlcTask Outputs/GVL_iXlinker.EtherCAT_Master_EJxxxx.Beckhoff_EJx9xx.A_0009_EJ2918_0000_0017.Module_2_FSOUT.Outputs.Module_2_Channel_2_Standard_Output <-> Module 2 (FSOUT)/Outputs/Module 2.Channel 2.Standard Output
//     PlcTask Outputs/GVL_iXlinker.EtherCAT_Master_EJxxxx.Beckhoff_EJx9xx.A_0009_EJ2918_0000_0017.Module_2_FSOUT.Outputs.Module_2_Channel_3_Standard_Output <-> Module 2 (FSOUT)/Outputs/Module 2.Channel 3.Standard Output
//     PlcTask Outputs/GVL_iXlinker.EtherCAT_Master_EJxxxx.Beckhoff_EJx9xx.A_0009_EJ2918_0000_0017.Module_2_FSOUT.Outputs.Module_2_Channel_4_Standard_Output <-> Module 2 (FSOUT)/Outputs/Module 2.Channel 4.Standard Output
//     PlcTask Inputs/GVL_iXlinker.EtherCAT_Master_EJxxxx.Beckhoff_EJx9xx.A_0009_EJ2918_0000_0017.Module_3_DEVICEIO.FIELDVOLTAGE_Field_Voltage_Status.Fieldvoltage_Underrange <-> Module 3 (DEVICEIO)/FIELDVOLTAGE Field Voltage Status/Fieldvoltage Underrange
//     PlcTask Inputs/GVL_iXlinker.EtherCAT_Master_EJxxxx.Beckhoff_EJx9xx.A_0009_EJ2918_0000_0017.Module_3_DEVICEIO.FIELDVOLTAGE_Field_Voltage_Status.Fieldvoltage_Overrange <-> Module 3 (DEVICEIO)/FIELDVOLTAGE Field Voltage Status/Fieldvoltage Overrange
//     PlcTask Inputs/GVL_iXlinker.EtherCAT_Master_EJxxxx.Beckhoff_EJx9xx.A_0009_EJ2918_0000_0017.Module_4_FSLOGIC.FSLOGIC_Inputs.Safe_Logic_State <-> Module 4 (FSLOGIC)/FSLOGIC Inputs/Safe Logic State
//     PlcTask Inputs/GVL_iXlinker.EtherCAT_Master_EJxxxx.Beckhoff_EJx9xx.A_0009_EJ2918_0000_0017.Module_4_FSLOGIC.FSLOGIC_Inputs.Cycle_Counter <-> Module 4 (FSLOGIC)/FSLOGIC Inputs/Cycle Counter
//     PlcTask Inputs/GVL_iXlinker.EtherCAT_Master_EJxxxx.Beckhoff_EJx9xx.A_0009_EJ2918_0000_0017.WcState.WcState0 <-> WcState/WcState0
//     PlcTask Inputs/GVL_iXlinker.EtherCAT_Master_EJxxxx.Beckhoff_EJx9xx.A_0009_EJ2918_0000_0017.WcState.WcState1 <-> WcState/WcState1
//     PlcTask Inputs/GVL_iXlinker.EtherCAT_Master_EJxxxx.Beckhoff_EJx9xx.A_0009_EJ2918_0000_0017.WcState.InputToggle0 <-> WcState/InputToggle0
//     PlcTask Inputs/GVL_iXlinker.EtherCAT_Master_EJxxxx.Beckhoff_EJx9xx.A_0009_EJ2918_0000_0017.WcState.InputToggle1 <-> WcState/InputToggle1
//     PlcTask Inputs/GVL_iXlinker.EtherCAT_Master_EJxxxx.Beckhoff_EJx9xx.A_0009_EJ2918_0000_0017.InfoData.AdsAddr <-> InfoData/AdsAddr
//     PlcTask Inputs/GVL_iXlinker.EtherCAT_Master_EJxxxx.Beckhoff_EJx9xx.A_0009_EJ2918_0000_0017.InfoData.State <-> InfoData/State
//   PLC/PLC Instance <-> EtherCAT Master EJxxxx/Beckhoff EJx9xx/A_0010(EJ2918-0000-0018)
//     PlcTask Inputs/GVL_iXlinker.EtherCAT_Master_EJxxxx.Beckhoff_EJx9xx.A_0010_EJ2918_0000_0018.Module_1_FSOE.FSoE_Inputs.FSOE/FSoE_Command <-> Module 1 (FSOE)/FSoE Inputs/FSOE/FSoE Command
//     PlcTask Inputs/GVL_iXlinker.EtherCAT_Master_EJxxxx.Beckhoff_EJx9xx.A_0010_EJ2918_0000_0018.Module_1_FSOE.FSoE_Inputs.FSOE/FSOUT_Module_1_Module_Fault <-> Module 1 (FSOE)/FSoE Inputs/FSOE/FSOUT Module 1.Module Fault
//     PlcTask Inputs/GVL_iXlinker.EtherCAT_Master_EJxxxx.Beckhoff_EJx9xx.A_0010_EJ2918_0000_0018.Module_1_FSOE.FSoE_Inputs.FSOE/FSOUT_Module_2_Module_Fault <-> Module 1 (FSOE)/FSoE Inputs/FSOE/FSOUT Module 2.Module Fault
//     PlcTask Inputs/GVL_iXlinker.EtherCAT_Master_EJxxxx.Beckhoff_EJx9xx.A_0010_EJ2918_0000_0018.Module_1_FSOE.FSoE_Inputs.FSOE/FSoE_CRC_000 <-> Module 1 (FSOE)/FSoE Inputs/FSOE/FSoE CRC 000
//     PlcTask Inputs/GVL_iXlinker.EtherCAT_Master_EJxxxx.Beckhoff_EJx9xx.A_0010_EJ2918_0000_0018.Module_1_FSOE.FSoE_Inputs.FSOE/FSoE_Connection_ID <-> Module 1 (FSOE)/FSoE Inputs/FSOE/FSoE Connection ID
//     PlcTask Outputs/GVL_iXlinker.EtherCAT_Master_EJxxxx.Beckhoff_EJx9xx.A_0010_EJ2918_0000_0018.Module_1_FSOE.FSoE_Outputs.FSOE/FSoE_Command <-> Module 1 (FSOE)/FSoE Outputs/FSOE/FSoE Command
//     PlcTask Outputs/GVL_iXlinker.EtherCAT_Master_EJxxxx.Beckhoff_EJx9xx.A_0010_EJ2918_0000_0018.Module_1_FSOE.FSoE_Outputs.FSOE/FSOUT_Module_1_Channel_1_Output <-> Module 1 (FSOE)/FSoE Outputs/FSOE/FSOUT Module 1.Channel 1.Output
//     PlcTask Outputs/GVL_iXlinker.EtherCAT_Master_EJxxxx.Beckhoff_EJx9xx.A_0010_EJ2918_0000_0018.Module_1_FSOE.FSoE_Outputs.FSOE/FSOUT_Module_1_Channel_2_Output <-> Module 1 (FSOE)/FSoE Outputs/FSOE/FSOUT Module 1.Channel 2.Output
//     PlcTask Outputs/GVL_iXlinker.EtherCAT_Master_EJxxxx.Beckhoff_EJx9xx.A_0010_EJ2918_0000_0018.Module_1_FSOE.FSoE_Outputs.FSOE/FSOUT_Module_1_Channel_3_Output <-> Module 1 (FSOE)/FSoE Outputs/FSOE/FSOUT Module 1.Channel 3.Output
//     PlcTask Outputs/GVL_iXlinker.EtherCAT_Master_EJxxxx.Beckhoff_EJx9xx.A_0010_EJ2918_0000_0018.Module_1_FSOE.FSoE_Outputs.FSOE/FSOUT_Module_1_Channel_4_Output <-> Module 1 (FSOE)/FSoE Outputs/FSOE/FSOUT Module 1.Channel 4.Output
//     PlcTask Outputs/GVL_iXlinker.EtherCAT_Master_EJxxxx.Beckhoff_EJx9xx.A_0010_EJ2918_0000_0018.Module_1_FSOE.FSoE_Outputs.FSOE/FSOUT_Module_2_Channel_1_Output <-> Module 1 (FSOE)/FSoE Outputs/FSOE/FSOUT Module 2.Channel 1.Output
//     PlcTask Outputs/GVL_iXlinker.EtherCAT_Master_EJxxxx.Beckhoff_EJx9xx.A_0010_EJ2918_0000_0018.Module_1_FSOE.FSoE_Outputs.FSOE/FSOUT_Module_2_Channel_2_Output <-> Module 1 (FSOE)/FSoE Outputs/FSOE/FSOUT Module 2.Channel 2.Output
//     PlcTask Outputs/GVL_iXlinker.EtherCAT_Master_EJxxxx.Beckhoff_EJx9xx.A_0010_EJ2918_0000_0018.Module_1_FSOE.FSoE_Outputs.FSOE/FSOUT_Module_2_Channel_3_Output <-> Module 1 (FSOE)/FSoE Outputs/FSOE/FSOUT Module 2.Channel 3.Output
//     PlcTask Outputs/GVL_iXlinker.EtherCAT_Master_EJxxxx.Beckhoff_EJx9xx.A_0010_EJ2918_0000_0018.Module_1_FSOE.FSoE_Outputs.FSOE/FSOUT_Module_2_Channel_4_Output <-> Module 1 (FSOE)/FSoE Outputs/FSOE/FSOUT Module 2.Channel 4.Output
//     PlcTask Outputs/GVL_iXlinker.EtherCAT_Master_EJxxxx.Beckhoff_EJx9xx.A_0010_EJ2918_0000_0018.Module_1_FSOE.FSoE_Outputs.FSOE/FSOUT_Module_1_ErrAck <-> Module 1 (FSOE)/FSoE Outputs/FSOE/FSOUT Module 1.ErrAck
//     PlcTask Outputs/GVL_iXlinker.EtherCAT_Master_EJxxxx.Beckhoff_EJx9xx.A_0010_EJ2918_0000_0018.Module_1_FSOE.FSoE_Outputs.FSOE/FSOUT_Module_2_ErrAck <-> Module 1 (FSOE)/FSoE Outputs/FSOE/FSOUT Module 2.ErrAck
//     PlcTask Outputs/GVL_iXlinker.EtherCAT_Master_EJxxxx.Beckhoff_EJx9xx.A_0010_EJ2918_0000_0018.Module_1_FSOE.FSoE_Outputs.FSOE/FSoE_CRC_000 <-> Module 1 (FSOE)/FSoE Outputs/FSOE/FSoE CRC 000
//     PlcTask Outputs/GVL_iXlinker.EtherCAT_Master_EJxxxx.Beckhoff_EJx9xx.A_0010_EJ2918_0000_0018.Module_1_FSOE.FSoE_Outputs.FSOE/FSoE_Connection_ID <-> Module 1 (FSOE)/FSoE Outputs/FSOE/FSoE Connection ID
//     PlcTask Outputs/GVL_iXlinker.EtherCAT_Master_EJxxxx.Beckhoff_EJx9xx.A_0010_EJ2918_0000_0018.Module_2_FSOUT.Outputs.Module_1_Channel_1_Standard_Output <-> Module 2 (FSOUT)/Outputs/Module 1.Channel 1.Standard Output
//     PlcTask Outputs/GVL_iXlinker.EtherCAT_Master_EJxxxx.Beckhoff_EJx9xx.A_0010_EJ2918_0000_0018.Module_2_FSOUT.Outputs.Module_1_Channel_2_Standard_Output <-> Module 2 (FSOUT)/Outputs/Module 1.Channel 2.Standard Output
//     PlcTask Outputs/GVL_iXlinker.EtherCAT_Master_EJxxxx.Beckhoff_EJx9xx.A_0010_EJ2918_0000_0018.Module_2_FSOUT.Outputs.Module_1_Channel_3_Standard_Output <-> Module 2 (FSOUT)/Outputs/Module 1.Channel 3.Standard Output
//     PlcTask Outputs/GVL_iXlinker.EtherCAT_Master_EJxxxx.Beckhoff_EJx9xx.A_0010_EJ2918_0000_0018.Module_2_FSOUT.Outputs.Module_1_Channel_4_Standard_Output <-> Module 2 (FSOUT)/Outputs/Module 1.Channel 4.Standard Output
//     PlcTask Outputs/GVL_iXlinker.EtherCAT_Master_EJxxxx.Beckhoff_EJx9xx.A_0010_EJ2918_0000_0018.Module_2_FSOUT.Outputs.Module_2_Channel_1_Standard_Output <-> Module 2 (FSOUT)/Outputs/Module 2.Channel 1.Standard Output
//     PlcTask Outputs/GVL_iXlinker.EtherCAT_Master_EJxxxx.Beckhoff_EJx9xx.A_0010_EJ2918_0000_0018.Module_2_FSOUT.Outputs.Module_2_Channel_2_Standard_Output <-> Module 2 (FSOUT)/Outputs/Module 2.Channel 2.Standard Output
//     PlcTask Outputs/GVL_iXlinker.EtherCAT_Master_EJxxxx.Beckhoff_EJx9xx.A_0010_EJ2918_0000_0018.Module_2_FSOUT.Outputs.Module_2_Channel_3_Standard_Output <-> Module 2 (FSOUT)/Outputs/Module 2.Channel 3.Standard Output
//     PlcTask Outputs/GVL_iXlinker.EtherCAT_Master_EJxxxx.Beckhoff_EJx9xx.A_0010_EJ2918_0000_0018.Module_2_FSOUT.Outputs.Module_2_Channel_4_Standard_Output <-> Module 2 (FSOUT)/Outputs/Module 2.Channel 4.Standard Output
//     PlcTask Inputs/GVL_iXlinker.EtherCAT_Master_EJxxxx.Beckhoff_EJx9xx.A_0010_EJ2918_0000_0018.Module_3_DEVICEIO.FIELDVOLTAGE_Field_Voltage_Status.Fieldvoltage_Underrange <-> Module 3 (DEVICEIO)/FIELDVOLTAGE Field Voltage Status/Fieldvoltage Underrange
//     PlcTask Inputs/GVL_iXlinker.EtherCAT_Master_EJxxxx.Beckhoff_EJx9xx.A_0010_EJ2918_0000_0018.Module_3_DEVICEIO.FIELDVOLTAGE_Field_Voltage_Status.Fieldvoltage_Overrange <-> Module 3 (DEVICEIO)/FIELDVOLTAGE Field Voltage Status/Fieldvoltage Overrange
//     PlcTask Inputs/GVL_iXlinker.EtherCAT_Master_EJxxxx.Beckhoff_EJx9xx.A_0010_EJ2918_0000_0018.Module_4_FSLOGIC.FSLOGIC_Inputs.Safe_Logic_State <-> Module 4 (FSLOGIC)/FSLOGIC Inputs/Safe Logic State
//     PlcTask Inputs/GVL_iXlinker.EtherCAT_Master_EJxxxx.Beckhoff_EJx9xx.A_0010_EJ2918_0000_0018.Module_4_FSLOGIC.FSLOGIC_Inputs.Cycle_Counter <-> Module 4 (FSLOGIC)/FSLOGIC Inputs/Cycle Counter
//     PlcTask Inputs/GVL_iXlinker.EtherCAT_Master_EJxxxx.Beckhoff_EJx9xx.A_0010_EJ2918_0000_0018.WcState.WcState0 <-> WcState/WcState0
//     PlcTask Inputs/GVL_iXlinker.EtherCAT_Master_EJxxxx.Beckhoff_EJx9xx.A_0010_EJ2918_0000_0018.WcState.WcState1 <-> WcState/WcState1
//     PlcTask Inputs/GVL_iXlinker.EtherCAT_Master_EJxxxx.Beckhoff_EJx9xx.A_0010_EJ2918_0000_0018.WcState.InputToggle0 <-> WcState/InputToggle0
//     PlcTask Inputs/GVL_iXlinker.EtherCAT_Master_EJxxxx.Beckhoff_EJx9xx.A_0010_EJ2918_0000_0018.WcState.InputToggle1 <-> WcState/InputToggle1
//     PlcTask Inputs/GVL_iXlinker.EtherCAT_Master_EJxxxx.Beckhoff_EJx9xx.A_0010_EJ2918_0000_0018.InfoData.AdsAddr <-> InfoData/AdsAddr
//     PlcTask Inputs/GVL_iXlinker.EtherCAT_Master_EJxxxx.Beckhoff_EJx9xx.A_0010_EJ2918_0000_0018.InfoData.State <-> InfoData/State
//   PLC/PLC Instance <-> EtherCAT Master EJxxxx/Beckhoff EJx9xx/A_0011(EJ6910-0000-0018)
//     PlcTask Inputs/GVL_iXlinker.EtherCAT_Master_EJxxxx.Beckhoff_EJx9xx.A_0011_EJ6910_0000_0018.FSLOGIC_Inputs.Safe_Logic_State <-> FSLOGIC Inputs/Safe Logic State
//     PlcTask Inputs/GVL_iXlinker.EtherCAT_Master_EJxxxx.Beckhoff_EJx9xx.A_0011_EJ6910_0000_0018.FSLOGIC_Inputs.Cycle_Counter <-> FSLOGIC Inputs/Cycle Counter
//     PlcTask Inputs/GVL_iXlinker.EtherCAT_Master_EJxxxx.Beckhoff_EJx9xx.A_0011_EJ6910_0000_0018.WcState.WcState <-> WcState/WcState
//     PlcTask Inputs/GVL_iXlinker.EtherCAT_Master_EJxxxx.Beckhoff_EJx9xx.A_0011_EJ6910_0000_0018.WcState.InputToggle <-> WcState/InputToggle
//     PlcTask Inputs/GVL_iXlinker.EtherCAT_Master_EJxxxx.Beckhoff_EJx9xx.A_0011_EJ6910_0000_0018.InfoData.AdsAddr <-> InfoData/AdsAddr
//     PlcTask Inputs/GVL_iXlinker.EtherCAT_Master_EJxxxx.Beckhoff_EJx9xx.A_0011_EJ6910_0000_0018.InfoData.State <-> InfoData/State
//   PLC/PLC Instance <-> EtherCAT Master EJxxxx/Beckhoff EJx9xx/A_0012(EJ6910-0000-0020)
//     PlcTask Inputs/GVL_iXlinker.EtherCAT_Master_EJxxxx.Beckhoff_EJx9xx.A_0012_EJ6910_0000_0020.FSLOGIC_Inputs.Safe_Logic_State <-> FSLOGIC Inputs/Safe Logic State
//     PlcTask Inputs/GVL_iXlinker.EtherCAT_Master_EJxxxx.Beckhoff_EJx9xx.A_0012_EJ6910_0000_0020.FSLOGIC_Inputs.Cycle_Counter <-> FSLOGIC Inputs/Cycle Counter
//     PlcTask Inputs/GVL_iXlinker.EtherCAT_Master_EJxxxx.Beckhoff_EJx9xx.A_0012_EJ6910_0000_0020.WcState.WcState <-> WcState/WcState
//     PlcTask Inputs/GVL_iXlinker.EtherCAT_Master_EJxxxx.Beckhoff_EJx9xx.A_0012_EJ6910_0000_0020.WcState.InputToggle <-> WcState/InputToggle
//     PlcTask Inputs/GVL_iXlinker.EtherCAT_Master_EJxxxx.Beckhoff_EJx9xx.A_0012_EJ6910_0000_0020.InfoData.AdsAddr <-> InfoData/AdsAddr
//     PlcTask Inputs/GVL_iXlinker.EtherCAT_Master_EJxxxx.Beckhoff_EJx9xx.A_0012_EJ6910_0000_0020.InfoData.State <-> InfoData/State
//   PLC/PLC Instance <-> EtherCAT_Master_EJxxxx
//     PlcTask Inputs/GVL_iXlinker.EtherCAT_Master_EJxxxx.SyncUnits._default._unreferenced.WcState.WcState <-> SyncUnits/<default>/<unreferenced>/WcState/WcState
//     PlcTask Inputs/GVL_iXlinker.EtherCAT_Master_EJxxxx.SyncUnits._default._unreferenced.InfoData.ObjectId <-> SyncUnits/<default>/<unreferenced>/InfoData/ObjectId
//     PlcTask Inputs/GVL_iXlinker.EtherCAT_Master_EJxxxx.SyncUnits._default._unreferenced.InfoData.State <-> SyncUnits/<default>/<unreferenced>/InfoData/State
//     PlcTask Inputs/GVL_iXlinker.EtherCAT_Master_EJxxxx.SyncUnits._default._unreferenced.InfoData.SlaveCount <-> SyncUnits/<default>/<unreferenced>/InfoData/SlaveCount
//     PlcTask Inputs/GVL_iXlinker.EtherCAT_Master_EJxxxx.SyncUnits._default.PlcTask.WcState.WcState <-> SyncUnits/<default>/PlcTask/WcState/WcState
//     PlcTask Inputs/GVL_iXlinker.EtherCAT_Master_EJxxxx.SyncUnits._default.PlcTask.InfoData.ObjectId <-> SyncUnits/<default>/PlcTask/InfoData/ObjectId
//     PlcTask Inputs/GVL_iXlinker.EtherCAT_Master_EJxxxx.SyncUnits._default.PlcTask.InfoData.State <-> SyncUnits/<default>/PlcTask/InfoData/State
//     PlcTask Inputs/GVL_iXlinker.EtherCAT_Master_EJxxxx.SyncUnits._default.PlcTask.InfoData.SlaveCount <-> SyncUnits/<default>/PlcTask/InfoData/SlaveCount
//     PlcTask Inputs/GVL_iXlinker.EtherCAT_Master_EJxxxx.Inputs.SlaveCount <-> Inputs/SlaveCount
//     PlcTask Inputs/GVL_iXlinker.EtherCAT_Master_EJxxxx.Inputs.DevState <-> Inputs/DevState
//     PlcTask Inputs/GVL_iXlinker.EtherCAT_Master_EJxxxx.Inputs.Frm{0..25}State <-> Inputs/Frm{0..25}State  (26 links)
//     PlcTask Inputs/GVL_iXlinker.EtherCAT_Master_EJxxxx.Inputs.Frm{0..25}WcState <-> Inputs/Frm{0..25}WcState  (26 links)
//     PlcTask Inputs/GVL_iXlinker.EtherCAT_Master_EJxxxx.Inputs.Frm{0..25}InputToggle <-> Inputs/Frm{0..25}InputToggle  (26 links)
//     PlcTask Outputs/GVL_iXlinker.EtherCAT_Master_EJxxxx.Outputs.DevCtrl <-> Outputs/DevCtrl
//     PlcTask Outputs/GVL_iXlinker.EtherCAT_Master_EJxxxx.Outputs.Frm{0..25}Ctrl <-> Outputs/Frm{0..25}Ctrl  (26 links)
//     PlcTask Outputs/GVL_iXlinker.EtherCAT_Master_EJxxxx.Outputs.Frm{0..25}WcCtrl <-> Outputs/Frm{0..25}WcCtrl  (26 links)
//     PlcTask Inputs/GVL_iXlinker.EtherCAT_Master_EJxxxx.InfoData.ChangeCount <-> InfoData/ChangeCount
//     PlcTask Inputs/GVL_iXlinker.EtherCAT_Master_EJxxxx.InfoData.DevId <-> InfoData/DevId
//     PlcTask Inputs/GVL_iXlinker.EtherCAT_Master_EJxxxx.InfoData.AmsNetId <-> InfoData/AmsNetId
//     PlcTask Inputs/GVL_iXlinker.EtherCAT_Master_EJxxxx.InfoData.CfgSlaveCount <-> InfoData/CfgSlaveCount
//     PlcTask Inputs/GVL_iXlinker.EtherCAT_Master_EJxxxx.InfoData.DcToTcTimeOffset <-> InfoData/DcToTcTimeOffset
//     PlcTask Inputs/GVL_iXlinker.EtherCAT_Master_EJxxxx.InfoData.DcToExtTimeOffset <-> InfoData/DcToExtTimeOffset

CONFIGURATION PLC
    RESOURCE PLC ON TwinCAT3
        TASK PlcTask(INTERVAL := T#10ms, PRIORITY := 20);
        PROGRAM MAIN WITH PlcTask : MAIN;
    END_RESOURCE
END_CONFIGURATION

// ---- DUTs/IO/PdoEntries/Status_B8381171.TcDUT
{attribute 'GeneratedUsingTerminal: EJ2521-0224-0016'}
{attribute addProperty BoxType "EJ2521-0224-0016"}
{attribute addProperty Id "Sel_Ack_End_counterBOOL1Ramp_activeBOOL1ErrorBOOL1Sync_errorBOOL1TxPDO_ToggleBOOL1"}
{attribute addProperty CRC "3090682225"}
{attribute addProperty Size "5"}
TYPE Status_B8381171 :
STRUCT
	{attribute addProperty Name "Sel_Ack_End_counter"}
	Sel_Ack_End_counter : BOOL;
	{attribute addProperty Name "Ramp_active"}
	Ramp_active : BOOL;
	{attribute addProperty Name "Error"}
	Error : BOOL;
	{attribute addProperty Name "Sync_error"}
	Sync_error : BOOL;
	{attribute addProperty Name "TxPDO_Toggle"}
	TxPDO_Toggle : BOOL;
END_STRUCT
END_TYPE

// ---- DUTs/IO/PdoEntries/Status_182674C6.TcDUT
{attribute 'GeneratedUsingTerminal: EJ2521-0224-0016'}
{attribute addProperty BoxType "EJ2521-0224-0016"}
{attribute addProperty Id "Latch_extern_validBOOL1Set_counter_doneBOOL1Counter_underflowBOOL1Counter_overflowBOOL1Status_of_extern_latchBOOL1Sync_errorBOOL1TxPDO_ToggleBOOL1"}
{attribute addProperty CRC "405173446"}
{attribute addProperty Size "7"}
TYPE Status_182674C6 :
STRUCT
	{attribute addProperty Name "Latch_extern_valid"}
	Latch_extern_valid : BOOL;
	{attribute addProperty Name "Set_counter_done"}
	Set_counter_done : BOOL;
	{attribute addProperty Name "Counter_underflow"}
	Counter_underflow : BOOL;
	{attribute addProperty Name "Counter_overflow"}
	Counter_overflow : BOOL;
	{attribute addProperty Name "Status_of_extern_latch"}
	Status_of_extern_latch : BOOL;
	{attribute addProperty Name "Sync_error"}
	Sync_error : BOOL;
	{attribute addProperty Name "TxPDO_Toggle"}
	TxPDO_Toggle : BOOL;
END_STRUCT
END_TYPE

// ---- DUTs/IO/PdoEntries/Status_7097155E.TcDUT
{attribute 'GeneratedUsingTerminal: EJ2521-0224-0016'}
{attribute addProperty BoxType "EJ2521-0224-0016"}
{attribute addProperty Id "PLS_EnabledBOOL1Status_of_outputBOOL1Sync_errorBOOL1TxPDO_ToggleBOOL1"}
{attribute addProperty CRC "1888949598"}
{attribute addProperty Size "4"}
TYPE Status_7097155E :
STRUCT
	{attribute addProperty Name "PLS_Enabled"}
	PLS_Enabled : BOOL;
	{attribute addProperty Name "Status_of_output"}
	Status_of_output : BOOL;
	{attribute addProperty Name "Sync_error"}
	Sync_error : BOOL;
	{attribute addProperty Name "TxPDO_Toggle"}
	TxPDO_Toggle : BOOL;
END_STRUCT
END_TYPE

// ---- DUTs/IO/PdoEntries/Control_DAEE1D52.TcDUT
{attribute 'GeneratedUsingTerminal: EJ2521-0224-0016'}
{attribute addProperty BoxType "EJ2521-0224-0016"}
{attribute addProperty Id "Frequency_selectBOOL1Disable_rampBOOL1Go_counterBOOL1"}
{attribute addProperty CRC "3673038162"}
{attribute addProperty Size "3"}
TYPE Control_DAEE1D52 :
STRUCT
	{attribute addProperty Name "Frequency_select"}
	Frequency_select : BOOL;
	{attribute addProperty Name "Disable_ramp"}
	Disable_ramp : BOOL;
	{attribute addProperty Name "Go_counter"}
	Go_counter : BOOL;
END_STRUCT
END_TYPE

// ---- DUTs/IO/PdoEntries/Control_F189B737.TcDUT
{attribute 'GeneratedUsingTerminal: EJ2521-0224-0016'}
{attribute addProperty BoxType "EJ2521-0224-0016"}
{attribute addProperty Id "Enable_latch_extern_on_positive_edgeBOOL1Set_counterBOOL1Enable_latch_extern_on_negative_edgeBOOL1"}
{attribute addProperty CRC "4052334391"}
{attribute addProperty Size "3"}
TYPE Control_F189B737 :
STRUCT
	{attribute addProperty Name "Enable_latch_extern_on_positive_edge"}
	Enable_latch_extern_on_positive_edge : BOOL;
	{attribute addProperty Name "Set_counter"}
	Set_counter : BOOL;
	{attribute addProperty Name "Enable_latch_extern_on_negative_edge"}
	Enable_latch_extern_on_negative_edge : BOOL;
END_STRUCT
END_TYPE

// ---- DUTs/IO/PdoEntries/Control_7786EF9F.TcDUT
{attribute 'GeneratedUsingTerminal: EJ2521-0224-0016'}
{attribute addProperty BoxType "EJ2521-0224-0016"}
{attribute addProperty Id "Enable_PLSBOOL1OutputBOOL1"}
{attribute addProperty CRC "2005331871"}
{attribute addProperty Size "2"}
TYPE Control_7786EF9F :
STRUCT
	{attribute addProperty Name "Enable_PLS"}
	Enable_PLS : BOOL;
	{attribute addProperty Name "Output"}
	Output : BOOL;
END_STRUCT
END_TYPE

// ---- DUTs/IO/PdoEntries/Status_70E023F8.TcDUT
{attribute 'GeneratedUsingTerminal: EJ2522-0000-0022'}
{attribute addProperty BoxType "EJ2522-0000-0022"}
{attribute addProperty Id "Set_counter_doneBOOL1Counter_underflowBOOL1Counter_overflowBOOL1Sync_errorBOOL1TxPDO_StateBOOL1TxPDO_ToggleBOOL1"}
{attribute addProperty CRC "1893737464"}
{attribute addProperty Size "6"}
TYPE Status_70E023F8 :
STRUCT
	{attribute addProperty Name "Set_counter_done"}
	Set_counter_done : BOOL;
	{attribute addProperty Name "Counter_underflow"}
	Counter_underflow : BOOL;
	{attribute addProperty Name "Counter_overflow"}
	Counter_overflow : BOOL;
	{attribute addProperty Name "Sync_error"}
	Sync_error : BOOL;
	{attribute addProperty Name "TxPDO_State"}
	TxPDO_State : BOOL;
	{attribute addProperty Name "TxPDO_Toggle"}
	TxPDO_Toggle : BOOL;
END_STRUCT
END_TYPE

// ---- DUTs/IO/PdoEntries/Control_A8DDCD82.TcDUT
{attribute 'GeneratedUsingTerminal: EJ2522-0000-0022'}
{attribute addProperty BoxType "EJ2522-0000-0022"}
{attribute addProperty Id "Set_counterBOOL1ReservedBOOL1"}
{attribute addProperty CRC "2833108354"}
{attribute addProperty Size "2"}
TYPE Control_A8DDCD82 :
STRUCT
	{attribute addProperty Name "Set_counter"}
	Set_counter : BOOL;
	{attribute addProperty Name "Reserved"}
	Reserved : BOOL;
END_STRUCT
END_TYPE

// ---- DUTs/IO/PdoEntries/Status_F2CE6D91.TcDUT
{attribute 'GeneratedUsingTerminal: EJ3004-0000-0019'}
{attribute addProperty BoxType "EJ3004-0000-0019"}
{attribute addProperty Id "UnderrangeBOOL1OverrangeBOOL1Limit_1BYTE1Limit_2BYTE1ErrorBOOL1TxPDO_StateBOOL1TxPDO_ToggleBOOL1"}
{attribute addProperty CRC "4073614737"}
{attribute addProperty Size "7"}
TYPE Status_F2CE6D91 :
STRUCT
	{attribute addProperty Name "Underrange"}
	Underrange : BOOL;
	{attribute addProperty Name "Overrange"}
	Overrange : BOOL;
	{attribute addProperty Name "Limit_1"}
	Limit_1 : BYTE;
	{attribute addProperty Name "Limit_2"}
	Limit_2 : BYTE;
	{attribute addProperty Name "Error"}
	Error : BOOL;
	{attribute addProperty Name "TxPDO_State"}
	TxPDO_State : BOOL;
	{attribute addProperty Name "TxPDO_Toggle"}
	TxPDO_Toggle : BOOL;
END_STRUCT
END_TYPE

// ---- DUTs/IO/PdoEntries/Status_B0753356.TcDUT
{attribute 'GeneratedUsingTerminal: EJ3104-0000-0019'}
{attribute addProperty BoxType "EJ3104-0000-0019"}
{attribute addProperty Id "UnderrangeBOOL1OverrangeBOOL1Limit_1BYTE1Limit_2BYTE1ErrorBOOL1Sync_errorBOOL1TxPDO_StateBOOL1TxPDO_ToggleBOOL1"}
{attribute addProperty CRC "2960470870"}
{attribute addProperty Size "8"}
TYPE Status_B0753356 :
STRUCT
	{attribute addProperty Name "Underrange"}
	Underrange : BOOL;
	{attribute addProperty Name "Overrange"}
	Overrange : BOOL;
	{attribute addProperty Name "Limit_1"}
	Limit_1 : BYTE;
	{attribute addProperty Name "Limit_2"}
	Limit_2 : BYTE;
	{attribute addProperty Name "Error"}
	Error : BOOL;
	{attribute addProperty Name "Sync_error"}
	Sync_error : BOOL;
	{attribute addProperty Name "TxPDO_State"}
	TxPDO_State : BOOL;
	{attribute addProperty Name "TxPDO_Toggle"}
	TxPDO_Toggle : BOOL;
END_STRUCT
END_TYPE

// ---- DUTs/IO/PdoEntries/Status_68C33E99.TcDUT
{attribute 'GeneratedUsingTerminal: EJ3214-0000-0016'}
{attribute addProperty BoxType "EJ3214-0000-0016"}
{attribute addProperty Id "UnderrangeBOOL1OverrangeBOOL1ErrorBOOL1TxPDO_StateBOOL1TxPDO_ToggleBOOL1"}
{attribute addProperty CRC "1757626009"}
{attribute addProperty Size "5"}
TYPE Status_68C33E99 :
STRUCT
	{attribute addProperty Name "Underrange"}
	Underrange : BOOL;
	{attribute addProperty Name "Overrange"}
	Overrange : BOOL;
	{attribute addProperty Name "Error"}
	Error : BOOL;
	{attribute addProperty Name "TxPDO_State"}
	TxPDO_State : BOOL;
	{attribute addProperty Name "TxPDO_Toggle"}
	TxPDO_Toggle : BOOL;
END_STRUCT
END_TYPE

// ---- DUTs/IO/PdoEntries/Status_ACC8459F.TcDUT
{attribute 'GeneratedUsingTerminal: EJ5002-0000-0016'}
{attribute addProperty BoxType "EJ5002-0000-0016"}
{attribute addProperty Id "Data_errorBOOL1Frame_errorBOOL1Power_failureBOOL1Sync_errorBOOL1TxPDO_StateBOOL1TxPDO_ToggleBOOL1"}
{attribute addProperty CRC "2898806175"}
{attribute addProperty Size "6"}
TYPE Status_ACC8459F :
STRUCT
	{attribute addProperty Name "Data_error"}
	Data_error : BOOL;
	{attribute addProperty Name "Frame_error"}
	Frame_error : BOOL;
	{attribute addProperty Name "Power_failure"}
	Power_failure : BOOL;
	{attribute addProperty Name "Sync_error"}
	Sync_error : BOOL;
	{attribute addProperty Name "TxPDO_State"}
	TxPDO_State : BOOL;
	{attribute addProperty Name "TxPDO_Toggle"}
	TxPDO_Toggle : BOOL;
END_STRUCT
END_TYPE

// ---- DUTs/IO/PdoEntries/Status_C03E2495.TcDUT
{attribute 'GeneratedUsingTerminal: EJ5002-0000-0017'}
{attribute addProperty BoxType "EJ5002-0000-0017"}
{attribute addProperty Id "Data_errorBOOL1Frame_errorBOOL1Power_failureBOOL1Data_mismatchBOOL1Sync_errorBOOL1TxPDO_StateBOOL1TxPDO_ToggleBOOL1"}
{attribute addProperty CRC "3225298069"}
{attribute addProperty Size "7"}
TYPE Status_C03E2495 :
STRUCT
	{attribute addProperty Name "Data_error"}
	Data_error : BOOL;
	{attribute addProperty Name "Frame_error"}
	Frame_error : BOOL;
	{attribute addProperty Name "Power_failure"}
	Power_failure : BOOL;
	{attribute addProperty Name "Data_mismatch"}
	Data_mismatch : BOOL;
	{attribute addProperty Name "Sync_error"}
	Sync_error : BOOL;
	{attribute addProperty Name "TxPDO_State"}
	TxPDO_State : BOOL;
	{attribute addProperty Name "TxPDO_Toggle"}
	TxPDO_Toggle : BOOL;
END_STRUCT
END_TYPE

// ---- DUTs/IO/PdoEntries/Status_D8D782C3.TcDUT
{attribute 'GeneratedUsingTerminal: EJ5101-0000-0016'}
{attribute addProperty BoxType "EJ5101-0000-0016"}
{attribute addProperty Id "Latch_C_validBOOL1Latch_extern_validBOOL1Set_counter_doneBOOL1Counter_underflowBOOL1Counter_overflowBOOL1Status_of_input_statusBOOL1Open_circuitBOOL1Extrapolation_stallBOOL1Status_of_input_ABOOL1Status_of_input_BBOOL1Status_of_input_CBOOL1Status_of_input_gateBOOL1Status_of_extern_latchBOOL1Sync_errorBOOL1TxPDO_StateBOOL1TxPDO_ToggleBOOL1"}
{attribute addProperty CRC "3638002371"}
{attribute addProperty Size "16"}
TYPE Status_D8D782C3 :
STRUCT
	{attribute addProperty Name "Latch_C_valid"}
	Latch_C_valid : BOOL;
	{attribute addProperty Name "Latch_extern_valid"}
	Latch_extern_valid : BOOL;
	{attribute addProperty Name "Set_counter_done"}
	Set_counter_done : BOOL;
	{attribute addProperty Name "Counter_underflow"}
	Counter_underflow : BOOL;
	{attribute addProperty Name "Counter_overflow"}
	Counter_overflow : BOOL;
	{attribute addProperty Name "Status_of_input_status"}
	Status_of_input_status : BOOL;
	{attribute addProperty Name "Open_circuit"}
	Open_circuit : BOOL;
	{attribute addProperty Name "Extrapolation_stall"}
	Extrapolation_stall : BOOL;
	{attribute addProperty Name "Status_of_input_A"}
	Status_of_input_A : BOOL;
	{attribute addProperty Name "Status_of_input_B"}
	Status_of_input_B : BOOL;
	{attribute addProperty Name "Status_of_input_C"}
	Status_of_input_C : BOOL;
	{attribute addProperty Name "Status_of_input_gate"}
	Status_of_input_gate : BOOL;
	{attribute addProperty Name "Status_of_extern_latch"}
	Status_of_extern_latch : BOOL;
	{attribute addProperty Name "Sync_error"}
	Sync_error : BOOL;
	{attribute addProperty Name "TxPDO_State"}
	TxPDO_State : BOOL;
	{attribute addProperty Name "TxPDO_Toggle"}
	TxPDO_Toggle : BOOL;
END_STRUCT
END_TYPE

// ---- DUTs/IO/PdoEntries/Control_6EF2C5D0.TcDUT
{attribute 'GeneratedUsingTerminal: EJ5101-0000-0016'}
{attribute addProperty BoxType "EJ5101-0000-0016"}
{attribute addProperty Id "Enable_latch_CBOOL1Enable_latch_extern_on_positive_edgeBOOL1Set_counterBOOL1Enable_latch_extern_on_negative_edgeBOOL1"}
{attribute addProperty CRC "1861404112"}
{attribute addProperty Size "4"}
TYPE Control_6EF2C5D0 :
STRUCT
	{attribute addProperty Name "Enable_latch_C"}
	Enable_latch_C : BOOL;
	{attribute addProperty Name "Enable_latch_extern_on_positive_edge"}
	Enable_latch_extern_on_positive_edge : BOOL;
	{attribute addProperty Name "Set_counter"}
	Set_counter : BOOL;
	{attribute addProperty Name "Enable_latch_extern_on_negative_edge"}
	Enable_latch_extern_on_negative_edge : BOOL;
END_STRUCT
END_TYPE

// ---- DUTs/IO/PdoEntries/Status_3E6F3FF3.TcDUT
{attribute 'GeneratedUsingTerminal: EJ5151-0000-0016'}
{attribute addProperty BoxType "EJ5151-0000-0016"}
{attribute addProperty Id "Latch_C_validBOOL1Latch_extern_validBOOL1Set_counter_doneBOOL1Extrapolation_stallBOOL1Status_of_input_ABOOL1Status_of_input_BBOOL1Status_of_input_CBOOL1Status_of_extern_latchBOOL1Sync_errorBOOL1TxPDO_ToggleBOOL1"}
{attribute addProperty CRC "1047478259"}
{attribute addProperty Size "10"}
TYPE Status_3E6F3FF3 :
STRUCT
	{attribute addProperty Name "Latch_C_valid"}
	Latch_C_valid : BOOL;
	{attribute addProperty Name "Latch_extern_valid"}
	Latch_extern_valid : BOOL;
	{attribute addProperty Name "Set_counter_done"}
	Set_counter_done : BOOL;
	{attribute addProperty Name "Extrapolation_stall"}
	Extrapolation_stall : BOOL;
	{attribute addProperty Name "Status_of_input_A"}
	Status_of_input_A : BOOL;
	{attribute addProperty Name "Status_of_input_B"}
	Status_of_input_B : BOOL;
	{attribute addProperty Name "Status_of_input_C"}
	Status_of_input_C : BOOL;
	{attribute addProperty Name "Status_of_extern_latch"}
	Status_of_extern_latch : BOOL;
	{attribute addProperty Name "Sync_error"}
	Sync_error : BOOL;
	{attribute addProperty Name "TxPDO_Toggle"}
	TxPDO_Toggle : BOOL;
END_STRUCT
END_TYPE

// ---- DUTs/IO/PdoEntries/Status_3D84275F.TcDUT
{attribute 'GeneratedUsingTerminal: EJ6002-0000-0016'}
{attribute addProperty BoxType "EJ6002-0000-0016"}
{attribute addProperty Id "Transmit_acceptedBOOL1Receive_requestBOOL1Init_acceptedBOOL1Buffer_fullBOOL1Parity_errorBOOL1Framing_errorBOOL1Overrun_errorBOOL1Input_lengthUSINT1"}
{attribute addProperty CRC "1032071007"}
{attribute addProperty Size "8"}
TYPE Status_3D84275F :
STRUCT
	{attribute addProperty Name "Transmit_accepted"}
	Transmit_accepted : BOOL;
	{attribute addProperty Name "Receive_request"}
	Receive_request : BOOL;
	{attribute addProperty Name "Init_accepted"}
	Init_accepted : BOOL;
	{attribute addProperty Name "Buffer_full"}
	Buffer_full : BOOL;
	{attribute addProperty Name "Parity_error"}
	Parity_error : BOOL;
	{attribute addProperty Name "Framing_error"}
	Framing_error : BOOL;
	{attribute addProperty Name "Overrun_error"}
	Overrun_error : BOOL;
	{attribute addProperty Name "Input_length"}
	Input_length : USINT;
END_STRUCT
END_TYPE

// ---- DUTs/IO/PdoEntries/Ctrl_1EFB4D3B.TcDUT
{attribute 'GeneratedUsingTerminal: EJ6002-0000-0016'}
{attribute addProperty BoxType "EJ6002-0000-0016"}
{attribute addProperty Id "Transmit_requestBOOL1Receive_acceptedBOOL1Init_requestBOOL1Send_continuousBOOL1Output_lengthUSINT1"}
{attribute addProperty CRC "519785787"}
{attribute addProperty Size "5"}
TYPE Ctrl_1EFB4D3B :
STRUCT
	{attribute addProperty Name "Transmit_request"}
	Transmit_request : BOOL;
	{attribute addProperty Name "Receive_accepted"}
	Receive_accepted : BOOL;
	{attribute addProperty Name "Init_request"}
	Init_request : BOOL;
	{attribute addProperty Name "Send_continuous"}
	Send_continuous : BOOL;
	{attribute addProperty Name "Output_length"}
	Output_length : USINT;
END_STRUCT
END_TYPE

// ---- DUTs/IO/PdoEntries/Status_B6795845.TcDUT
{attribute 'GeneratedUsingTerminal: EJ7031-0000-0026'}
{attribute addProperty BoxType "EJ7031-0000-0026"}
{attribute addProperty Id "Ready_to_enableBOOL1ReadyBOOL1WarningBOOL1ErrorBOOL1Moving_positiveBOOL1Moving_negativeBOOL1Torque_reducedBOOL1Digital_input_1BOOL1Digital_input_2BOOL1Sync_errorBOOL1TxPDO_ToggleBOOL1"}
{attribute addProperty CRC "3061405765"}
{attribute addProperty Size "11"}
TYPE Status_B6795845 :
STRUCT
	{attribute addProperty Name "Ready_to_enable"}
	Ready_to_enable : BOOL;
	{attribute addProperty Name "Ready"}
	Ready : BOOL;
	{attribute addProperty Name "Warning"}
	Warning : BOOL;
	{attribute addProperty Name "Error"}
	Error : BOOL;
	{attribute addProperty Name "Moving_positive"}
	Moving_positive : BOOL;
	{attribute addProperty Name "Moving_negative"}
	Moving_negative : BOOL;
	{attribute addProperty Name "Torque_reduced"}
	Torque_reduced : BOOL;
	{attribute addProperty Name "Digital_input_1"}
	Digital_input_1 : BOOL;
	{attribute addProperty Name "Digital_input_2"}
	Digital_input_2 : BOOL;
	{attribute addProperty Name "Sync_error"}
	Sync_error : BOOL;
	{attribute addProperty Name "TxPDO_Toggle"}
	TxPDO_Toggle : BOOL;
END_STRUCT
END_TYPE

// ---- DUTs/IO/PdoEntries/Control_C948E0F2.TcDUT
{attribute 'GeneratedUsingTerminal: EJ7031-0000-0026'}
{attribute addProperty BoxType "EJ7031-0000-0026"}
{attribute addProperty Id "EnableBOOL1ResetBOOL1Reduce_torqueBOOL1"}
{attribute addProperty CRC "3376996594"}
{attribute addProperty Size "3"}
TYPE Control_C948E0F2 :
STRUCT
	{attribute addProperty Name "Enable"}
	Enable : BOOL;
	{attribute addProperty Name "Reset"}
	Reset : BOOL;
	{attribute addProperty Name "Reduce_torque"}
	Reduce_torque : BOOL;
END_STRUCT
END_TYPE

// ---- DUTs/IO/PdoEntries/Status_8CBE219F.TcDUT
{attribute 'GeneratedUsingTerminal: EJ7037-0000-0020'}
{attribute addProperty BoxType "EJ7037-0000-0020"}
{attribute addProperty Id "Latch_C_validBOOL1Latch_extern_validBOOL1Set_counter_doneBOOL1Counter_underflowBOOL1Counter_overflowBOOL1Extrapolation_stallBOOL1Status_of_input_ABOOL1Status_of_input_BBOOL1Status_of_input_CBOOL1Status_of_extern_latchBOOL1Sync_errorBOOL1TxPDO_ToggleBOOL1"}
{attribute addProperty CRC "2361270687"}
{attribute addProperty Size "12"}
TYPE Status_8CBE219F :
STRUCT
	{attribute addProperty Name "Latch_C_valid"}
	Latch_C_valid : BOOL;
	{attribute addProperty Name "Latch_extern_valid"}
	Latch_extern_valid : BOOL;
	{attribute addProperty Name "Set_counter_done"}
	Set_counter_done : BOOL;
	{attribute addProperty Name "Counter_underflow"}
	Counter_underflow : BOOL;
	{attribute addProperty Name "Counter_overflow"}
	Counter_overflow : BOOL;
	{attribute addProperty Name "Extrapolation_stall"}
	Extrapolation_stall : BOOL;
	{attribute addProperty Name "Status_of_input_A"}
	Status_of_input_A : BOOL;
	{attribute addProperty Name "Status_of_input_B"}
	Status_of_input_B : BOOL;
	{attribute addProperty Name "Status_of_input_C"}
	Status_of_input_C : BOOL;
	{attribute addProperty Name "Status_of_extern_latch"}
	Status_of_extern_latch : BOOL;
	{attribute addProperty Name "Sync_error"}
	Sync_error : BOOL;
	{attribute addProperty Name "TxPDO_Toggle"}
	TxPDO_Toggle : BOOL;
END_STRUCT
END_TYPE

// ---- DUTs/IO/PdoEntries/Status_1E008DB9.TcDUT
{attribute 'GeneratedUsingTerminal: EJ7037-0000-0020'}
{attribute addProperty BoxType "EJ7037-0000-0020"}
{attribute addProperty Id "Ready_to_enableBOOL1ReadyBOOL1WarningBOOL1ErrorBOOL1Moving_positiveBOOL1Moving_negativeBOOL1Torque_reducedBOOL1Motor_stallBOOL1Digital_input_1BOOL1Digital_input_2BOOL1Sync_errorBOOL1TxPDO_ToggleBOOL1"}
{attribute addProperty CRC "503352761"}
{attribute addProperty Size "12"}
TYPE Status_1E008DB9 :
STRUCT
	{attribute addProperty Name "Ready_to_enable"}
	Ready_to_enable : BOOL;
	{attribute addProperty Name "Ready"}
	Ready : BOOL;
	{attribute addProperty Name "Warning"}
	Warning : BOOL;
	{attribute addProperty Name "Error"}
	Error : BOOL;
	{attribute addProperty Name "Moving_positive"}
	Moving_positive : BOOL;
	{attribute addProperty Name "Moving_negative"}
	Moving_negative : BOOL;
	{attribute addProperty Name "Torque_reduced"}
	Torque_reduced : BOOL;
	{attribute addProperty Name "Motor_stall"}
	Motor_stall : BOOL;
	{attribute addProperty Name "Digital_input_1"}
	Digital_input_1 : BOOL;
	{attribute addProperty Name "Digital_input_2"}
	Digital_input_2 : BOOL;
	{attribute addProperty Name "Sync_error"}
	Sync_error : BOOL;
	{attribute addProperty Name "TxPDO_Toggle"}
	TxPDO_Toggle : BOOL;
END_STRUCT
END_TYPE

// ---- DUTs/IO/PdoEntries/Control_5FD4673D.TcDUT
{attribute 'GeneratedUsingTerminal: EJ7037-0000-0020'}
{attribute addProperty BoxType "EJ7037-0000-0020"}
{attribute addProperty Id "EnableBOOL1ResetBOOL1Reduce_torqueBOOL1Digital_output_1BOOL1"}
{attribute addProperty CRC "1607755581"}
{attribute addProperty Size "4"}
TYPE Control_5FD4673D :
STRUCT
	{attribute addProperty Name "Enable"}
	Enable : BOOL;
	{attribute addProperty Name "Reset"}
	Reset : BOOL;
	{attribute addProperty Name "Reduce_torque"}
	Reduce_torque : BOOL;
	{attribute addProperty Name "Digital_output_1"}
	Digital_output_1 : BOOL;
END_STRUCT
END_TYPE

// ---- DUTs/IO/PdoEntries/Status_3035BE2E.TcDUT
{attribute 'GeneratedUsingTerminal: EJ7342-0000-0019'}
{attribute addProperty BoxType "EJ7342-0000-0019"}
{attribute addProperty Id "Latch_extern_validBOOL1Set_counter_doneBOOL1Counter_underflowBOOL1Counter_overflowBOOL1Extrapolation_stallBOOL1Status_of_input_ABOOL1Status_of_input_BBOOL1Status_of_extern_latchBOOL1Sync_errorBOOL1TxPDO_ToggleBOOL1"}
{attribute addProperty CRC "808828462"}
{attribute addProperty Size "10"}
TYPE Status_3035BE2E :
STRUCT
	{attribute addProperty Name "Latch_extern_valid"}
	Latch_extern_valid : BOOL;
	{attribute addProperty Name "Set_counter_done"}
	Set_counter_done : BOOL;
	{attribute addProperty Name "Counter_underflow"}
	Counter_underflow : BOOL;
	{attribute addProperty Name "Counter_overflow"}
	Counter_overflow : BOOL;
	{attribute addProperty Name "Extrapolation_stall"}
	Extrapolation_stall : BOOL;
	{attribute addProperty Name "Status_of_input_A"}
	Status_of_input_A : BOOL;
	{attribute addProperty Name "Status_of_input_B"}
	Status_of_input_B : BOOL;
	{attribute addProperty Name "Status_of_extern_latch"}
	Status_of_extern_latch : BOOL;
	{attribute addProperty Name "Sync_error"}
	Sync_error : BOOL;
	{attribute addProperty Name "TxPDO_Toggle"}
	TxPDO_Toggle : BOOL;
END_STRUCT
END_TYPE

// ---- DUTs/IO/PdoEntries/Status_2569232E.TcDUT
{attribute 'GeneratedUsingTerminal: EJ7334-0008-0016'}
{attribute addProperty BoxType "EJ7334-0008-0016"}
{attribute addProperty Id "Ready_to_enableBOOL1ReadyBOOL1WarningBOOL1ErrorBOOL1Moving_positiveBOOL1Moving_negativeBOOL1Limit_xBOOL1TxPDO_ToggleBOOL1"}
{attribute addProperty CRC "627647278"}
{attribute addProperty Size "8"}
TYPE Status_2569232E :
STRUCT
	{attribute addProperty Name "Ready_to_enable"}
	Ready_to_enable : BOOL;
	{attribute addProperty Name "Ready"}
	Ready : BOOL;
	{attribute addProperty Name "Warning"}
	Warning : BOOL;
	{attribute addProperty Name "Error"}
	Error : BOOL;
	{attribute addProperty Name "Moving_positive"}
	Moving_positive : BOOL;
	{attribute addProperty Name "Moving_negative"}
	Moving_negative : BOOL;
	{attribute addProperty Name "Limit_x"}
	Limit_x : BOOL;
	{attribute addProperty Name "TxPDO_Toggle"}
	TxPDO_Toggle : BOOL;
END_STRUCT
END_TYPE

